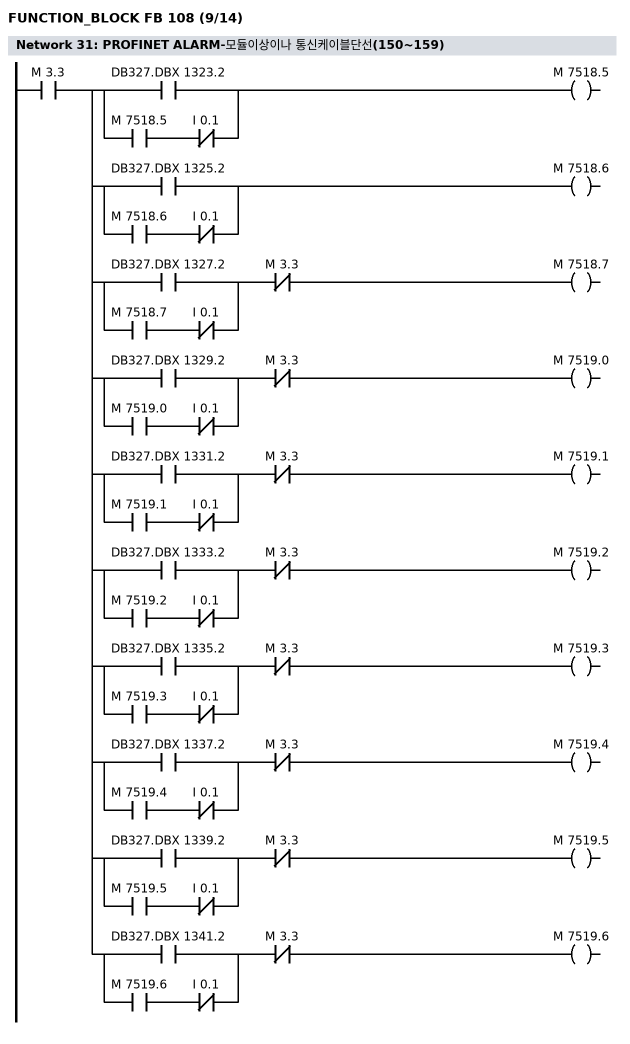

      A     M      3.3;
      =     L      0.0;
      A     L      0.0;
      A(    ;
      O     DB327.DBX 1323.2;
      O     ;
      A     M   7518.5;
      AN    I      0.1;
      )     ;
      =     M   7518.5;
      A     L      0.0;
      A(    ;
      O     DB327.DBX 1325.2;
      O     ;
      A     M   7518.6;
      AN    I      0.1;
      )     ;
      =     M   7518.6;
      A     L      0.0;
      A(    ;
      O     DB327.DBX 1327.2;
      O     ;
      A     M   7518.7;
      AN    I      0.1;
      )     ;
      AN    M      3.3;
      =     M   7518.7;
      A     L      0.0;
      A(    ;
      O     DB327.DBX 1329.2;
      O     ;
      A     M   7519.0;
      AN    I      0.1;
      )     ;
      AN    M      3.3;
      =     M   7519.0;
      A     L      0.0;
      A(    ;
      O     DB327.DBX 1331.2;
      O     ;
      A     M   7519.1;
      AN    I      0.1;
      )     ;
      AN    M      3.3;
      =     M   7519.1;
      A     L      0.0;
      A(    ;
      O     DB327.DBX 1333.2;
      O     ;
      A     M   7519.2;
      AN    I      0.1;
      )     ;
      AN    M      3.3;
      =     M   7519.2;
      A     L      0.0;
      A(    ;
      O     DB327.DBX 1335.2;
      O     ;
      A     M   7519.3;
      AN    I      0.1;
      )     ;
      AN    M      3.3;
      =     M   7519.3;
      A     L      0.0;
      A(    ;
      O     DB327.DBX 1337.2;
      O     ;
      A     M   7519.4;
      AN    I      0.1;
      )     ;
      AN    M      3.3;
      =     M   7519.4;
      A     L      0.0;
      A(    ;
      O     DB327.DBX 1339.2;
      O     ;
      A     M   7519.5;
      AN    I      0.1;
      )     ;
      AN    M      3.3;
      =     M   7519.5;
      A     L      0.0;
      A(    ;
      O     DB327.DBX 1341.2;
      O     ;
      A     M   7519.6;
      AN    I      0.1;
      )     ;
      AN    M      3.3;
      =     M   7519.6;
NETWORK
TITLE =PROFINET MODULE ERROR(1~10)
//
//
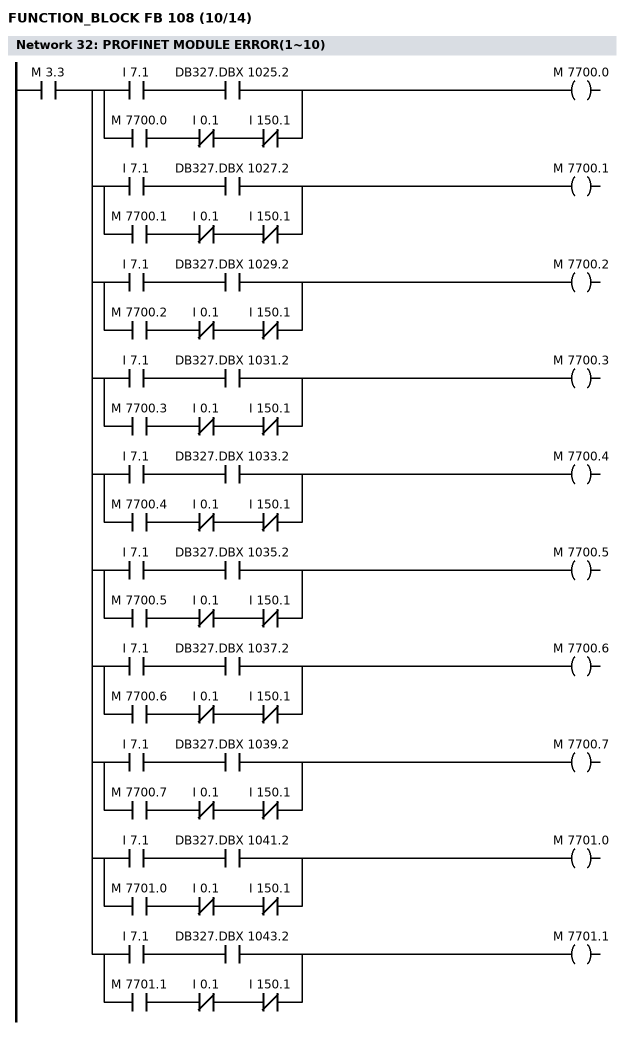
      A     M      3.3;
      =     L      0.0;
      A     L      0.0;
      A(    ;
      A     I      7.1;
      A     DB327.DBX 1025.2;
      O     ;
      A     M   7700.0;
      AN    I      0.1;
      AN    I    150.1;
      )     ;
      =     M   7700.0;
      A     L      0.0;
      A(    ;
      A     I      7.1;
      A     DB327.DBX 1027.2;
      O     ;
      A     M   7700.1;
      AN    I      0.1;
      AN    I    150.1;
      )     ;
      =     M   7700.1;
      A     L      0.0;
      A(    ;
      A     I      7.1;
      A     DB327.DBX 1029.2;
      O     ;
      A     M   7700.2;
      AN    I      0.1;
      AN    I    150.1;
      )     ;
      =     M   7700.2;
      A     L      0.0;
      A(    ;
      A     I      7.1;
      A     DB327.DBX 1031.2;
      O     ;
      A     M   7700.3;
      AN    I      0.1;
      AN    I    150.1;
      )     ;
      =     M   7700.3;
      A     L      0.0;
      A(    ;
      A     I      7.1;
      A     DB327.DBX 1033.2;
      O     ;
      A     M   7700.4;
      AN    I      0.1;
      AN    I    150.1;
      )     ;
      =     M   7700.4;
      A     L      0.0;
      A(    ;
      A     I      7.1;
      A     DB327.DBX 1035.2;
      O     ;
      A     M   7700.5;
      AN    I      0.1;
      AN    I    150.1;
      )     ;
      =     M   7700.5;
      A     L      0.0;
      A(    ;
      A     I      7.1;
      A     DB327.DBX 1037.2;
      O     ;
      A     M   7700.6;
      AN    I      0.1;
      AN    I    150.1;
      )     ;
      =     M   7700.6;
      A     L      0.0;
      A(    ;
      A     I      7.1;
      A     DB327.DBX 1039.2;
      O     ;
      A     M   7700.7;
      AN    I      0.1;
      AN    I    150.1;
      )     ;
      =     M   7700.7;
      A     L      0.0;
      A(    ;
      A     I      7.1;
      A     DB327.DBX 1041.2;
      O     ;
      A     M   7701.0;
      AN    I      0.1;
      AN    I    150.1;
      )     ;
      =     M   7701.0;
      A     L      0.0;
      A(    ;
      A     I      7.1;
      A     DB327.DBX 1043.2;
      O     ;
      A     M   7701.1;
      AN    I      0.1;
      AN    I    150.1;
      )     ;
      =     M   7701.1;
NETWORK
TITLE =PROFINET MODULE ERROR(11~20)
//
//
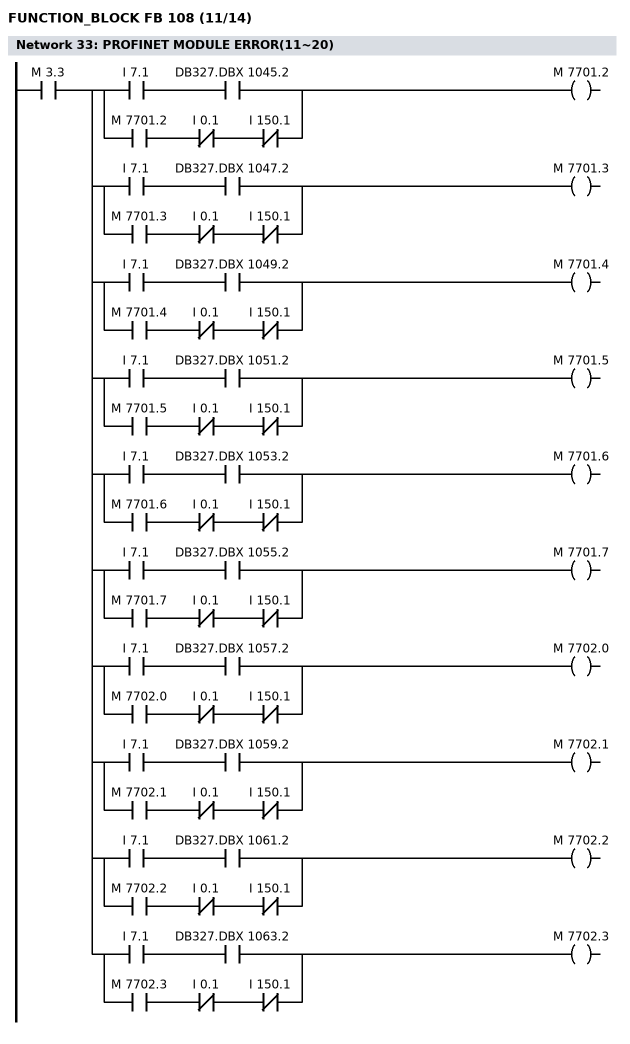
      A     M      3.3;
      =     L      0.0;
      A     L      0.0;
      A(    ;
      A     I      7.1;
      A     DB327.DBX 1045.2;
      O     ;
      A     M   7701.2;
      AN    I      0.1;
      AN    I    150.1;
      )     ;
      =     M   7701.2;
      A     L      0.0;
      A(    ;
      A     I      7.1;
      A     DB327.DBX 1047.2;
      O     ;
      A     M   7701.3;
      AN    I      0.1;
      AN    I    150.1;
      )     ;
      =     M   7701.3;
      A     L      0.0;
      A(    ;
      A     I      7.1;
      A     DB327.DBX 1049.2;
      O     ;
      A     M   7701.4;
      AN    I      0.1;
      AN    I    150.1;
      )     ;
      =     M   7701.4;
      A     L      0.0;
      A(    ;
      A     I      7.1;
      A     DB327.DBX 1051.2;
      O     ;
      A     M   7701.5;
      AN    I      0.1;
      AN    I    150.1;
      )     ;
      =     M   7701.5;
      A     L      0.0;
      A(    ;
      A     I      7.1;
      A     DB327.DBX 1053.2;
      O     ;
      A     M   7701.6;
      AN    I      0.1;
      AN    I    150.1;
      )     ;
      =     M   7701.6;
      A     L      0.0;
      A(    ;
      A     I      7.1;
      A     DB327.DBX 1055.2;
      O     ;
      A     M   7701.7;
      AN    I      0.1;
      AN    I    150.1;
      )     ;
      =     M   7701.7;
      A     L      0.0;
      A(    ;
      A     I      7.1;
      A     DB327.DBX 1057.2;
      O     ;
      A     M   7702.0;
      AN    I      0.1;
      AN    I    150.1;
      )     ;
      =     M   7702.0;
      A     L      0.0;
      A(    ;
      A     I      7.1;
      A     DB327.DBX 1059.2;
      O     ;
      A     M   7702.1;
      AN    I      0.1;
      AN    I    150.1;
      )     ;
      =     M   7702.1;
      A     L      0.0;
      A(    ;
      A     I      7.1;
      A     DB327.DBX 1061.2;
      O     ;
      A     M   7702.2;
      AN    I      0.1;
      AN    I    150.1;
      )     ;
      =     M   7702.2;
      A     L      0.0;
      A(    ;
      A     I      7.1;
      A     DB327.DBX 1063.2;
      O     ;
      A     M   7702.3;
      AN    I      0.1;
      AN    I    150.1;
      )     ;
      =     M   7702.3;
NETWORK
TITLE =PROFINET MODULE ERROR(21~30)
//
//
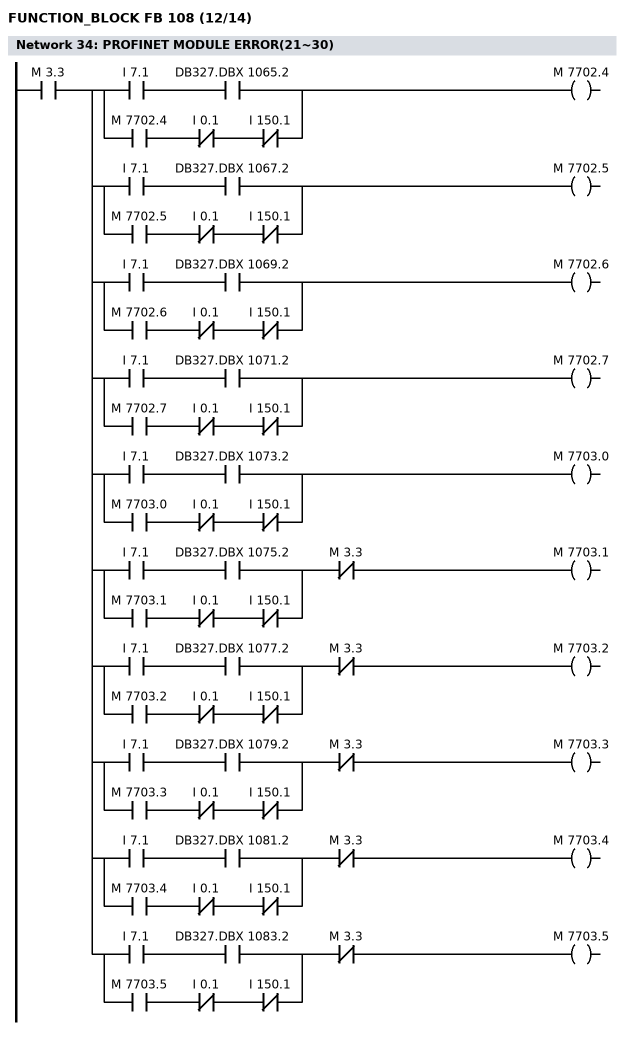
      A     M      3.3;
      =     L      0.0;
      A     L      0.0;
      A(    ;
      A     I      7.1;
      A     DB327.DBX 1065.2;
      O     ;
      A     M   7702.4;
      AN    I      0.1;
      AN    I    150.1;
      )     ;
      =     M   7702.4;
      A     L      0.0;
      A(    ;
      A     I      7.1;
      A     DB327.DBX 1067.2;
      O     ;
      A     M   7702.5;
      AN    I      0.1;
      AN    I    150.1;
      )     ;
      =     M   7702.5;
      A     L      0.0;
      A(    ;
      A     I      7.1;
      A     DB327.DBX 1069.2;
      O     ;
      A     M   7702.6;
      AN    I      0.1;
      AN    I    150.1;
      )     ;
      =     M   7702.6;
      A     L      0.0;
      A(    ;
      A     I      7.1;
      A     DB327.DBX 1071.2;
      O     ;
      A     M   7702.7;
      AN    I      0.1;
      AN    I    150.1;
      )     ;
      =     M   7702.7;
      A     L      0.0;
      A(    ;
      A     I      7.1;
      A     DB327.DBX 1073.2;
      O     ;
      A     M   7703.0;
      AN    I      0.1;
      AN    I    150.1;
      )     ;
      =     M   7703.0;
      A     L      0.0;
      A(    ;
      A     I      7.1;
      A     DB327.DBX 1075.2;
      O     ;
      A     M   7703.1;
      AN    I      0.1;
      AN    I    150.1;
      )     ;
      AN    M      3.3;
      =     M   7703.1;
      A     L      0.0;
      A(    ;
      A     I      7.1;
      A     DB327.DBX 1077.2;
      O     ;
      A     M   7703.2;
      AN    I      0.1;
      AN    I    150.1;
      )     ;
      AN    M      3.3;
      =     M   7703.2;
      A     L      0.0;
      A(    ;
      A     I      7.1;
      A     DB327.DBX 1079.2;
      O     ;
      A     M   7703.3;
      AN    I      0.1;
      AN    I    150.1;
      )     ;
      AN    M      3.3;
      =     M   7703.3;
      A     L      0.0;
      A(    ;
      A     I      7.1;
      A     DB327.DBX 1081.2;
      O     ;
      A     M   7703.4;
      AN    I      0.1;
      AN    I    150.1;
      )     ;
      AN    M      3.3;
      =     M   7703.4;
      A     L      0.0;
      A(    ;
      A     I      7.1;
      A     DB327.DBX 1083.2;
      O     ;
      A     M   7703.5;
      AN    I      0.1;
      AN    I    150.1;
      )     ;
      AN    M      3.3;
      =     M   7703.5;
NETWORK
TITLE =PROFINET MODULE ERROR(31~40)
//
//
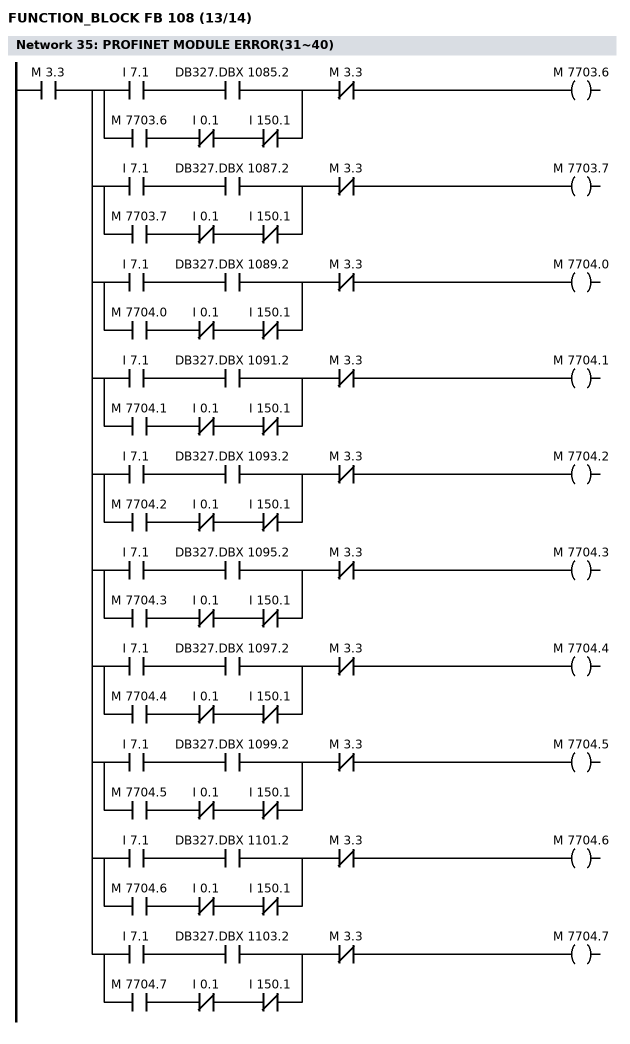
      A     M      3.3;
      =     L      0.0;
      A     L      0.0;
      A(    ;
      A     I      7.1;
      A     DB327.DBX 1085.2;
      O     ;
      A     M   7703.6;
      AN    I      0.1;
      AN    I    150.1;
      )     ;
      AN    M      3.3;
      =     M   7703.6;
      A     L      0.0;
      A(    ;
      A     I      7.1;
      A     DB327.DBX 1087.2;
      O     ;
      A     M   7703.7;
      AN    I      0.1;
      AN    I    150.1;
      )     ;
      AN    M      3.3;
      =     M   7703.7;
      A     L      0.0;
      A(    ;
      A     I      7.1;
      A     DB327.DBX 1089.2;
      O     ;
      A     M   7704.0;
      AN    I      0.1;
      AN    I    150.1;
      )     ;
      AN    M      3.3;
      =     M   7704.0;
      A     L      0.0;
      A(    ;
      A     I      7.1;
      A     DB327.DBX 1091.2;
      O     ;
      A     M   7704.1;
      AN    I      0.1;
      AN    I    150.1;
      )     ;
      AN    M      3.3;
      =     M   7704.1;
      A     L      0.0;
      A(    ;
      A     I      7.1;
      A     DB327.DBX 1093.2;
      O     ;
      A     M   7704.2;
      AN    I      0.1;
      AN    I    150.1;
      )     ;
      AN    M      3.3;
      =     M   7704.2;
      A     L      0.0;
      A(    ;
      A     I      7.1;
      A     DB327.DBX 1095.2;
      O     ;
      A     M   7704.3;
      AN    I      0.1;
      AN    I    150.1;
      )     ;
      AN    M      3.3;
      =     M   7704.3;
      A     L      0.0;
      A(    ;
      A     I      7.1;
      A     DB327.DBX 1097.2;
      O     ;
      A     M   7704.4;
      AN    I      0.1;
      AN    I    150.1;
      )     ;
      AN    M      3.3;
      =     M   7704.4;
      A     L      0.0;
      A(    ;
      A     I      7.1;
      A     DB327.DBX 1099.2;
      O     ;
      A     M   7704.5;
      AN    I      0.1;
      AN    I    150.1;
      )     ;
      AN    M      3.3;
      =     M   7704.5;
      A     L      0.0;
      A(    ;
      A     I      7.1;
      A     DB327.DBX 1101.2;
      O     ;
      A     M   7704.6;
      AN    I      0.1;
      AN    I    150.1;
      )     ;
      AN    M      3.3;
      =     M   7704.6;
      A     L      0.0;
      A(    ;
      A     I      7.1;
      A     DB327.DBX 1103.2;
      O     ;
      A     M   7704.7;
      AN    I      0.1;
      AN    I    150.1;
      )     ;
      AN    M      3.3;
      =     M   7704.7;
NETWORK
TITLE =PROFINET MODULE ERROR(150~159)
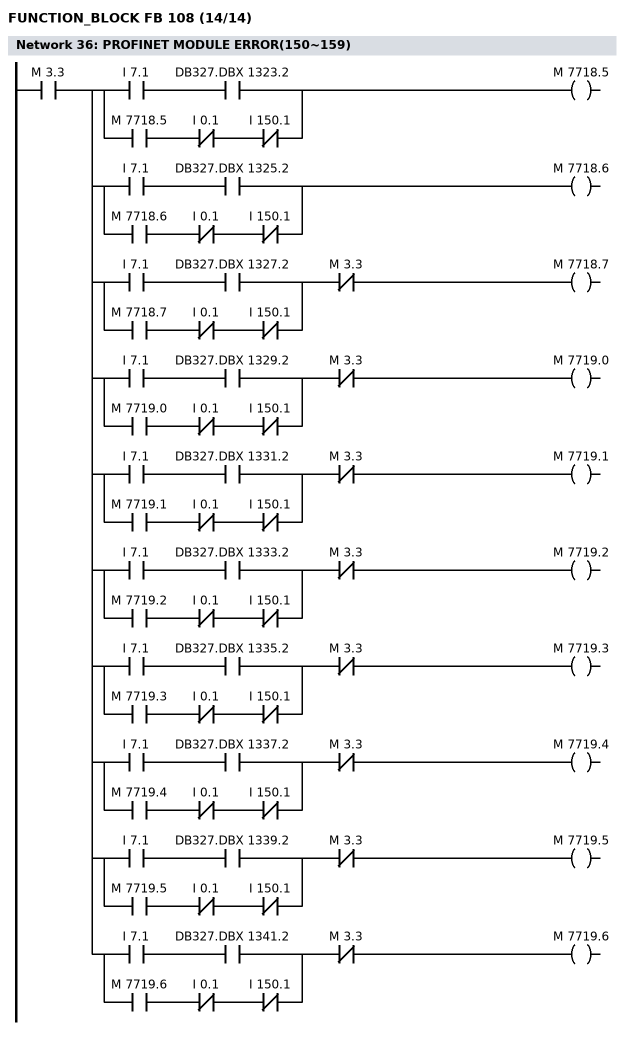

      A     M      3.3;
      =     L      0.0;
      A     L      0.0;
      A(    ;
      A     I      7.1;
      A     DB327.DBX 1323.2;
      O     ;
      A     M   7718.5;
      AN    I      0.1;
      AN    I    150.1;
      )     ;
      =     M   7718.5;
      A     L      0.0;
      A(    ;
      A     I      7.1;
      A     DB327.DBX 1325.2;
      O     ;
      A     M   7718.6;
      AN    I      0.1;
      AN    I    150.1;
      )     ;
      =     M   7718.6;
      A     L      0.0;
      A(    ;
      A     I      7.1;
      A     DB327.DBX 1327.2;
      O     ;
      A     M   7718.7;
      AN    I      0.1;
      AN    I    150.1;
      )     ;
      AN    M      3.3;
      =     M   7718.7;
      A     L      0.0;
      A(    ;
      A     I      7.1;
      A     DB327.DBX 1329.2;
      O     ;
      A     M   7719.0;
      AN    I      0.1;
      AN    I    150.1;
      )     ;
      AN    M      3.3;
      =     M   7719.0;
      A     L      0.0;
      A(    ;
      A     I      7.1;
      A     DB327.DBX 1331.2;
      O     ;
      A     M   7719.1;
      AN    I      0.1;
      AN    I    150.1;
      )     ;
      AN    M      3.3;
      =     M   7719.1;
      A     L      0.0;
      A(    ;
      A     I      7.1;
      A     DB327.DBX 1333.2;
      O     ;
      A     M   7719.2;
      AN    I      0.1;
      AN    I    150.1;
      )     ;
      AN    M      3.3;
      =     M   7719.2;
      A     L      0.0;
      A(    ;
      A     I      7.1;
      A     DB327.DBX 1335.2;
      O     ;
      A     M   7719.3;
      AN    I      0.1;
      AN    I    150.1;
      )     ;
      AN    M      3.3;
      =     M   7719.3;
      A     L      0.0;
      A(    ;
      A     I      7.1;
      A     DB327.DBX 1337.2;
      O     ;
      A     M   7719.4;
      AN    I      0.1;
      AN    I    150.1;
      )     ;
      AN    M      3.3;
      =     M   7719.4;
      A     L      0.0;
      A(    ;
      A     I      7.1;
      A     DB327.DBX 1339.2;
      O     ;
      A     M   7719.5;
      AN    I      0.1;
      AN    I    150.1;
      )     ;
      AN    M      3.3;
      =     M   7719.5;
      A     L      0.0;
      A(    ;
      A     I      7.1;
      A     DB327.DBX 1341.2;
      O     ;
      A     M   7719.6;
      AN    I      0.1;
      AN    I    150.1;
      )     ;
      AN    M      3.3;
      =     M   7719.6;
END_FUNCTION_BLOCK

DATA_BLOCK DB 108
TITLE =
VERSION : 0.0

 FB 108
BEGIN
END_DATA_BLOCK

FUNCTION FC 108 : VOID
TITLE =
VERSION : 0.1

BEGIN
NETWORK
TITLE =

      AN    OV;
      =     L      0.0;
      A     L      0.0;
      AN    M   1000.0;
      =     M   3800.0;
      A     L      0.0;
      AN    M   2500.0;
      =     M   3800.1;
      A     L      0.0;
      AN    I     16.0;
      =     M   3800.2;
      A     L      0.0;
      A     M    503.1;
      =     M   3800.3;
NETWORK
TITLE =

      AN    OV;
      =     L      0.0;
      A     L      0.0;
      A     M    503.3;
      =     M   3800.4;
      A     L      0.0;
      A     M    503.2;
      =     M   3800.5;
      A     L      0.0;
      A     M    503.2;
      =     M   3800.6;
      A     L      0.0;
      AN    I    100.7;
      =     M   3800.7;
NETWORK
TITLE =

      AN    OV;
      =     L      0.0;
      A     L      0.0;
      AN    I    100.3;
      =     M   3801.0;
      A     L      0.0;
      AN    I    100.1;
      =     M   3801.1;
      A     L      0.0;
      AN    I    100.6;
      =     M   3801.2;
      A     L      0.0;
      AN    I    100.4;
      =     M   3801.3;
NETWORK
TITLE =

      AN    OV;
      =     L      0.0;
      A     L      0.0;
      AN    I    100.0;
      =     M   3801.4;
      A     L      0.0;
      AN    I     29.5;
      =     M   3801.5;
      A     L      0.0;
      AN    I    129.1;
      =     M   3801.6;
      A     L      0.0;
      AN    I    100.2;
      =     M   3801.7;
NETWORK
TITLE =

      AN    OV;
      =     L      0.0;
      A     L      0.0;
      A     M   2503.4;
      =     M   3802.3;
      A     L      0.0;
      A     M   2503.5;
      =     M   3802.4;
      A     L      0.0;
      A     M   2503.6;
      =     M   3802.5;
      A     L      0.0;
      A     M   1003.6;
      =     M   3802.6;
      A     L      0.0;
      A     M   1004.2;
      =     M   3802.7;
NETWORK
TITLE =

      AN    OV;
      =     L      0.0;
      A     L      0.0;
      A     M   2504.2;
      =     M   3803.0;
      A     L      0.0;
      A(    ;
      O     M   2550.0;
      O     M   2550.1;
      )     ;
      =     M   3803.1;
      A     L      0.0;
      A(    ;
      O     M   2550.2;
      O     M   2550.3;
      )     ;
      =     M   3803.2;
      A     L      0.0;
      A(    ;
      O     M   2515.2;
      O     M   2550.4;
      O     M   2550.5;
      )     ;
      =     M   3803.3;
NETWORK
TITLE =

      AN    OV;
      =     L      0.0;
      A     L      0.0;
      A(    ;
      O     M   1050.0;
      O     M   1050.1;
      )     ;
      =     M   3803.4;
      A     L      0.0;
      A(    ;
      O     M   1050.2;
      O     M   1050.3;
      )     ;
      =     M   3803.5;
      A     L      0.0;
      A(    ;
      O     M   1050.4;
      O     M   1050.5;
      )     ;
      =     M   3803.6;
      A     L      0.0;
      A(    ;
      O     M   1050.6;
      O     M   1050.7;
      )     ;
      =     M   3803.7;
NETWORK
TITLE =

      AN    OV;
      =     L      0.0;
      A     L      0.0;
      A(    ;
      O     M   1051.0;
      O     M   1051.1;
      )     ;
      =     M   3804.0;
      A     L      0.0;
      A(    ;
      O     M   1051.2;
      O     M   1051.3;
      )     ;
      =     M   3804.1;
      A     L      0.0;
      A(    ;
      O     M   1051.4;
      O     M   1051.5;
      )     ;
      =     M   3804.2;
      A     L      0.0;
      A(    ;
      O     M   1051.6;
      O     M   1051.7;
      )     ;
      =     M   3804.3;
      A     L      0.0;
      A     M   5200.7;
      =     M   3805.5;
NETWORK
TITLE =
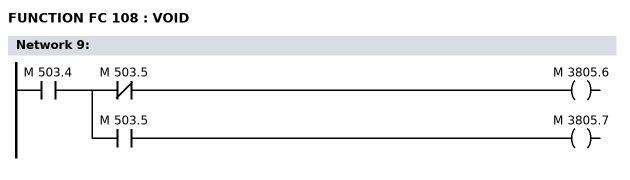

      A     M    503.4;
      =     L      0.0;
      A     L      0.0;
      AN    M    503.5;
      =     M   3805.6;
      A     L      0.0;
      A     M    503.5;
      =     M   3805.7;
NETWORK
TITLE =

      AN    OV;
      =     L      0.0;
      A     L      0.0;
      A(    ;
      O     I      2.1;
      O     I     49.6;
      O     T    134;
      )     ;
      =     M   3808.5;
      A     L      0.0;
      A     I      2.1;
      =     M   3808.6;
NETWORK
TITLE =
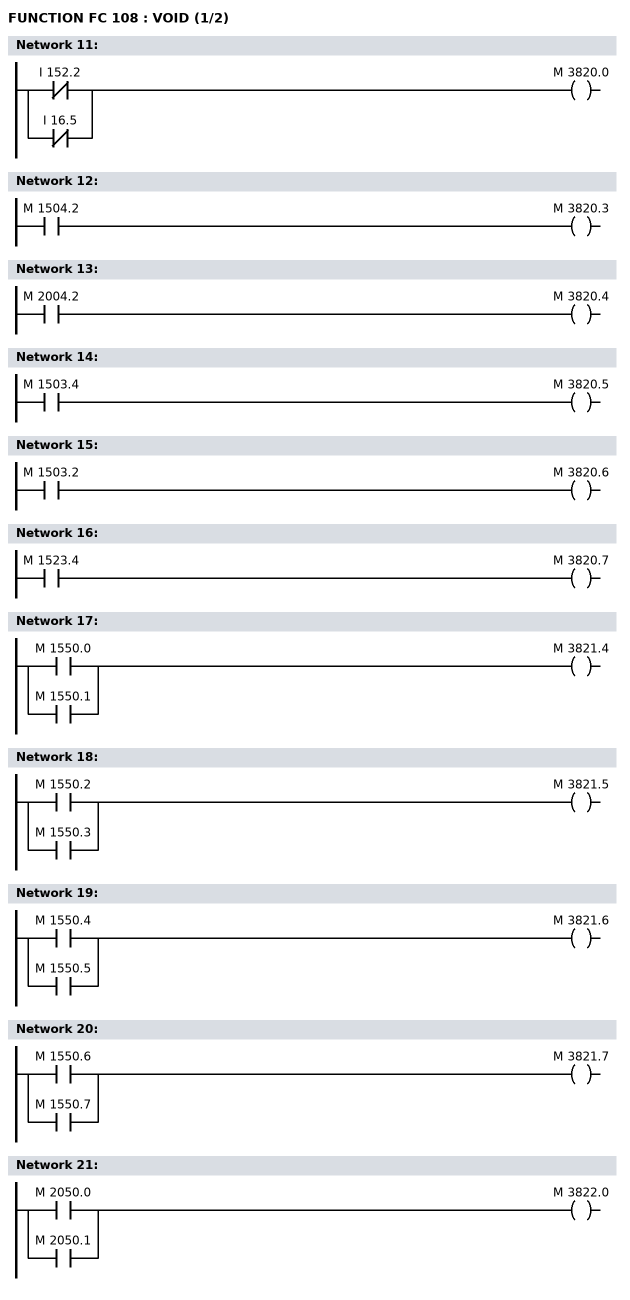

      ON    I    152.2;
      ON    I     16.5;
      =     M   3820.0;
NETWORK
TITLE =

      A     M   1504.2;
      =     M   3820.3;
NETWORK
TITLE =

      A     M   2004.2;
      =     M   3820.4;
NETWORK
TITLE =

      A     M   1503.4;
      =     M   3820.5;
NETWORK
TITLE =

      A     M   1503.2;
      =     M   3820.6;
NETWORK
TITLE =

      A     M   1523.4;
      =     M   3820.7;
NETWORK
TITLE =

      O     M   1550.0;
      O     M   1550.1;
      =     M   3821.4;
NETWORK
TITLE =

      O     M   1550.2;
      O     M   1550.3;
      =     M   3821.5;
NETWORK
TITLE =

      O     M   1550.4;
      O     M   1550.5;
      =     M   3821.6;
NETWORK
TITLE =

      O     M   1550.6;
      O     M   1550.7;
      =     M   3821.7;
NETWORK
TITLE =

      O     M   2050.0;
      O     M   2050.1;
      =     M   3822.0;
NETWORK
TITLE =
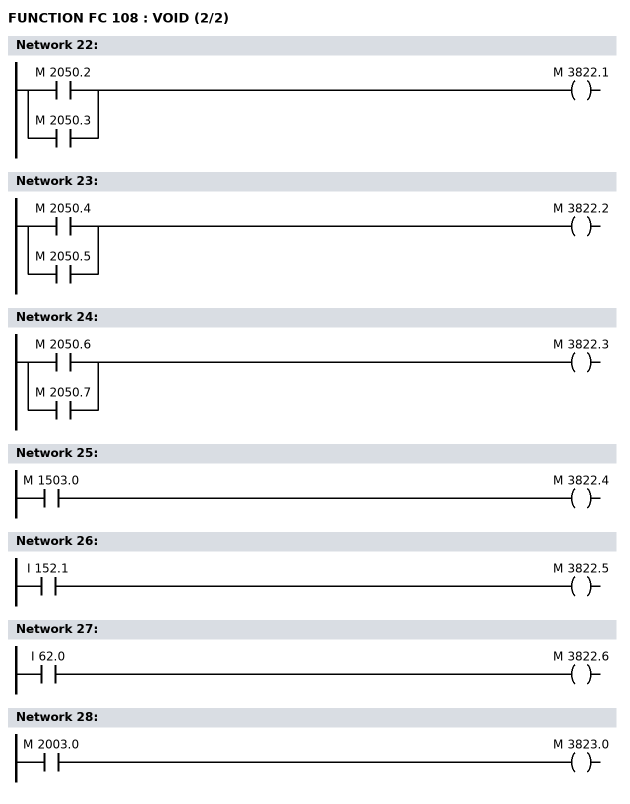

      O     M   2050.2;
      O     M   2050.3;
      =     M   3822.1;
NETWORK
TITLE =

      O     M   2050.4;
      O     M   2050.5;
      =     M   3822.2;
NETWORK
TITLE =

      O     M   2050.6;
      O     M   2050.7;
      =     M   3822.3;
NETWORK
TITLE =

      A     M   1503.0;
      =     M   3822.4;
NETWORK
TITLE =

      A     I    152.1;
      =     M   3822.5;
NETWORK
TITLE =

      A     I     62.0;
      =     M   3822.6;
NETWORK
TITLE =

      A     M   2003.0;
      =     M   3823.0;
NETWORK
TITLE =

      AN    OV;
      =     L      0.0;
      A     L      0.0;
      AN    I   1011.0;
      =     M   3824.0;
      A     L      0.0;
      A     I   1011.1;
      =     M   3824.1;
      A     L      0.0;
      A     I   1011.2;
      =     M   3824.2;
      A     L      0.0;
      A     I   1011.4;
      =     M   3824.3;
      A     L      0.0;
      A     I   1011.5;
      =     M   3824.4;
      A     L      0.0;
      A     I   1011.6;
      =     M   3824.5;
      A     L      0.0;
      A     I   1011.7;
      =     M   3824.6;
      A     L      0.0;
      A     I   1010.5;
      =     M   3824.7;
NETWORK
TITLE =

      AN    OV;
      =     L      0.0;
      A     L      0.0;
      AN    I   1019.0;
      =     M   3825.0;
      A     L      0.0;
      A     I   1019.1;
      =     M   3825.1;
      A     L      0.0;
      A     I   1019.2;
      =     M   3825.2;
      A     L      0.0;
      A     I   1019.4;
      =     M   3825.3;
      A     L      0.0;
      A     I   1019.5;
      =     M   3825.4;
      A     L      0.0;
      A     I   1019.6;
      =     M   3825.5;
      A     L      0.0;
      A     I   1019.7;
      =     M   3825.6;
      A     L      0.0;
      A     I   1018.5;
      =     M   3825.7;
NETWORK
TITLE =

      AN    OV;
      =     L      0.0;
      A     L      0.0;
      AN    I   1027.0;
      =     M   3826.0;
      A     L      0.0;
      A     I   1027.1;
      =     M   3826.1;
      A     L      0.0;
      A     I   1027.2;
      =     M   3826.2;
      A     L      0.0;
      A     I   1027.4;
      =     M   3826.3;
      A     L      0.0;
      A     I   1027.5;
      =     M   3826.4;
      A     L      0.0;
      A     I   1027.6;
      =     M   3826.5;
      A     L      0.0;
      A     I   1027.7;
      =     M   3826.6;
      A     L      0.0;
      A     I   1026.5;
      =     M   3826.7;
NETWORK
TITLE =

      AN    OV;
      =     L      0.0;
      A     L      0.0;
      AN    I   1035.0;
      =     M   3827.0;
      A     L      0.0;
      A     I   1035.1;
      =     M   3827.1;
      A     L      0.0;
      A     I   1035.2;
      =     M   3827.2;
      A     L      0.0;
      A     I   1035.4;
      =     M   3827.3;
      A     L      0.0;
      A     I   1035.5;
      =     M   3827.4;
      A     L      0.0;
      A     I   1035.6;
      =     M   3827.5;
      A     L      0.0;
      A     I   1035.7;
      =     M   3827.6;
      A     L      0.0;
      A     I   1034.5;
      =     M   3827.7;
NETWORK
TITLE =
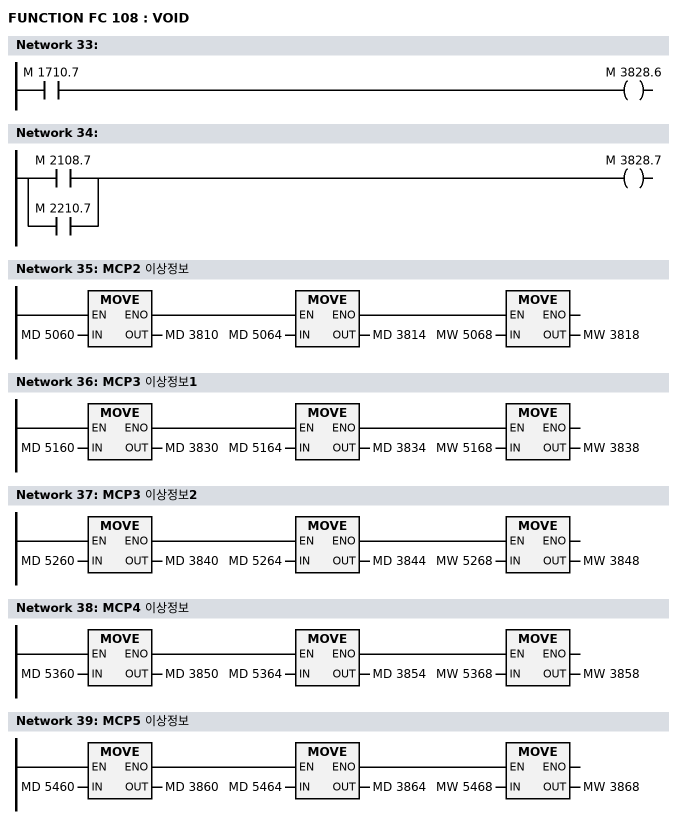

      A     M   1710.7;
      =     M   3828.6;
NETWORK
TITLE =

      O     M   2108.7;
      O     M   2210.7;
      =     M   3828.7;
NETWORK
TITLE =MCP2 이상정보

      A(    ;
      A(    ;
      L     MD  5060;
      T     MD  3810;
      SET   ;
      SAVE  ;
      CLR   ;
      A     BR;
      )     ;
      JNB   _001;
      L     MD  5064;
      T     MD  3814;
      SET   ;
      SAVE  ;
      CLR   ;
_001: A     BR;
      )     ;
      JNB   _002;
      L     MW  5068;
      T     MW  3818;
_002: NOP   0;
NETWORK
TITLE =MCP3 이상정보1

      A(    ;
      A(    ;
      L     MD  5160;
      T     MD  3830;
      SET   ;
      SAVE  ;
      CLR   ;
      A     BR;
      )     ;
      JNB   _003;
      L     MD  5164;
      T     MD  3834;
      SET   ;
      SAVE  ;
      CLR   ;
_003: A     BR;
      )     ;
      JNB   _004;
      L     MW  5168;
      T     MW  3838;
_004: NOP   0;
NETWORK
TITLE =MCP3 이상정보2

      A(    ;
      A(    ;
      L     MD  5260;
      T     MD  3840;
      SET   ;
      SAVE  ;
      CLR   ;
      A     BR;
      )     ;
      JNB   _005;
      L     MD  5264;
      T     MD  3844;
      SET   ;
      SAVE  ;
      CLR   ;
_005: A     BR;
      )     ;
      JNB   _006;
      L     MW  5268;
      T     MW  3848;
_006: NOP   0;
NETWORK
TITLE =MCP4 이상정보

      A(    ;
      A(    ;
      L     MD  5360;
      T     MD  3850;
      SET   ;
      SAVE  ;
      CLR   ;
      A     BR;
      )     ;
      JNB   _007;
      L     MD  5364;
      T     MD  3854;
      SET   ;
      SAVE  ;
      CLR   ;
_007: A     BR;
      )     ;
      JNB   _008;
      L     MW  5368;
      T     MW  3858;
_008: NOP   0;
NETWORK
TITLE =MCP5 이상정보

      A(    ;
      A(    ;
      L     MD  5460;
      T     MD  3860;
      SET   ;
      SAVE  ;
      CLR   ;
      A     BR;
      )     ;
      JNB   _009;
      L     MD  5464;
      T     MD  3864;
      SET   ;
      SAVE  ;
      CLR   ;
_009: A     BR;
      )     ;
      JNB   _00a;
      L     MW  5468;
      T     MW  3868;
_00a: NOP   0;
END_FUNCTION

FUNCTION FC 109 : VOID
TITLE =
VERSION : 0.1

BEGIN
NETWORK
TITLE =
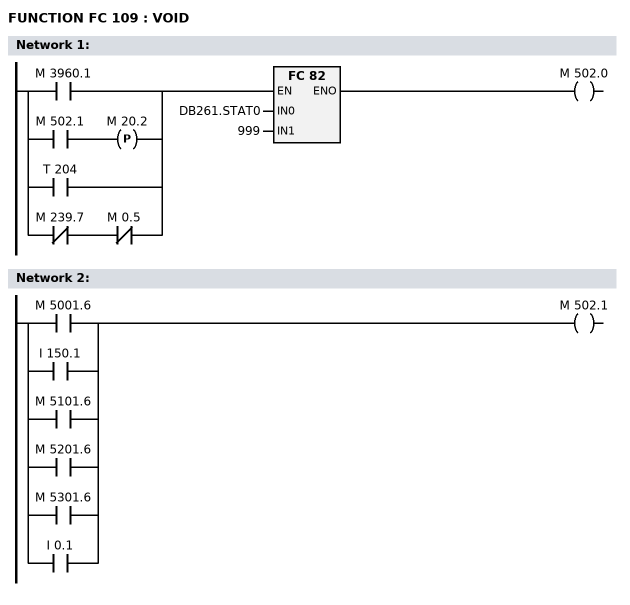

      A(    ;
      O     M   3960.1;
      O(    ;
      A     M    502.1;
      FP    M     20.2;
      )     ;
      O     T    204;
      O     ;
      AN    M    239.7;
      AN    M      0.5;
      )     ;
      JNB   _001;
      CALL FC    82 (
           IN0                      := DB261.STAT0,
           IN1                      := 999);
_001: A     BR;
      =     M    502.0;
NETWORK
TITLE =

      O     M   5001.6;
      O     I    150.1;
      O     M   5101.6;
      O     M   5201.6;
      O     M   5301.6;
      O     I      0.1;
      =     M    502.1;
NETWORK
TITLE =

      AN    OV;
      =     L      0.0;
      A     L      0.0;
      A     M    502.0;
      L     S5T#1S;
      SE    T    205;
      A     L      0.0;
      AN    M    239.7;
      L     S5T#1S;
      SD    T    203;
      A     L      0.0;
      A     T    203;
      L     S5T#1S;
      SE    T    204;
NETWORK
TITLE =
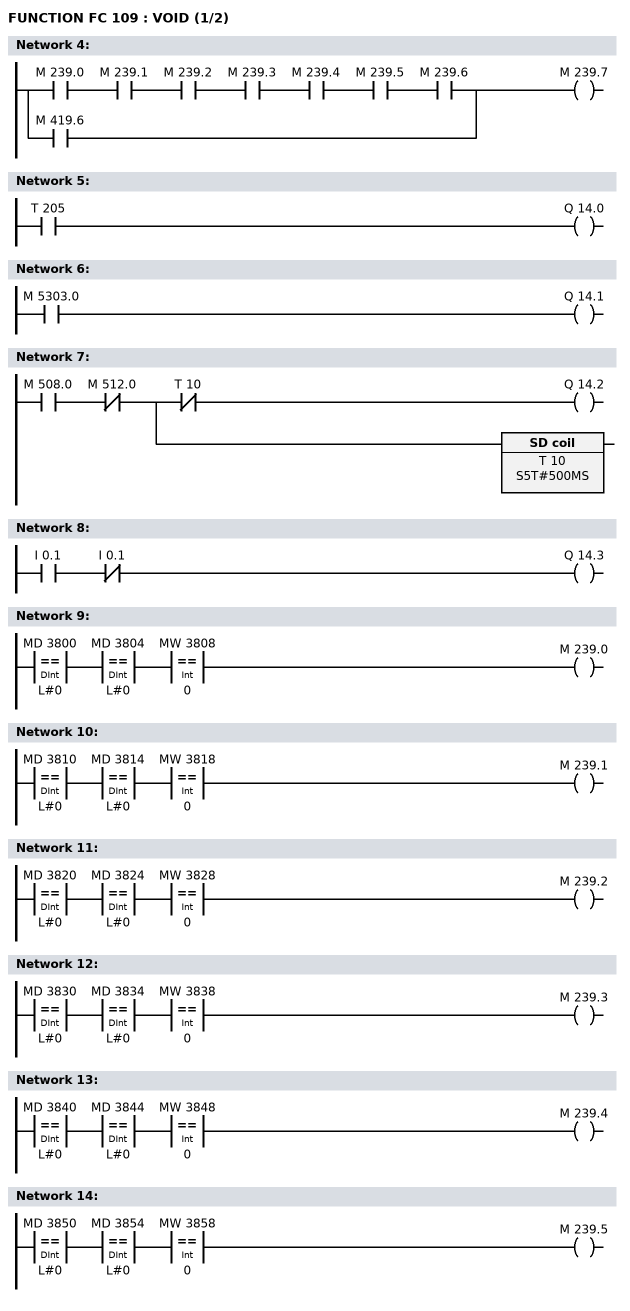

      A     M    239.0;
      A     M    239.1;
      A     M    239.2;
      A     M    239.3;
      A     M    239.4;
      A     M    239.5;
      A     M    239.6;
      O     M    419.6;
      =     M    239.7;
NETWORK
TITLE =

      A     T    205;
      =     Q     14.0;
NETWORK
TITLE =

      A     M   5303.0;
      =     Q     14.1;
NETWORK
TITLE =

      A     M    508.0;
      AN    M    512.0;
      =     L      0.0;
      A     L      0.0;
      AN    T     10;
      =     Q     14.2;
      A     L      0.0;
      BLD   102;
      L     S5T#500MS;
      SD    T     10;
NETWORK
TITLE =

      A     I      0.1;
      AN    I      0.1;
      =     Q     14.3;
NETWORK
TITLE =

      A(    ;
      L     MD  3800;
      L     L#0;
      ==D   ;
      )     ;
      A(    ;
      L     MD  3804;
      L     L#0;
      ==D   ;
      )     ;
      A(    ;
      L     MW  3808;
      L     0;
      ==I   ;
      )     ;
      =     M    239.0;
NETWORK
TITLE =

      A(    ;
      L     MD  3810;
      L     L#0;
      ==D   ;
      )     ;
      A(    ;
      L     MD  3814;
      L     L#0;
      ==D   ;
      )     ;
      A(    ;
      L     MW  3818;
      L     0;
      ==I   ;
      )     ;
      =     M    239.1;
NETWORK
TITLE =

      A(    ;
      L     MD  3820;
      L     L#0;
      ==D   ;
      )     ;
      A(    ;
      L     MD  3824;
      L     L#0;
      ==D   ;
      )     ;
      A(    ;
      L     MW  3828;
      L     0;
      ==I   ;
      )     ;
      =     M    239.2;
NETWORK
TITLE =

      A(    ;
      L     MD  3830;
      L     L#0;
      ==D   ;
      )     ;
      A(    ;
      L     MD  3834;
      L     L#0;
      ==D   ;
      )     ;
      A(    ;
      L     MW  3838;
      L     0;
      ==I   ;
      )     ;
      =     M    239.3;
NETWORK
TITLE =

      A(    ;
      L     MD  3840;
      L     L#0;
      ==D   ;
      )     ;
      A(    ;
      L     MD  3844;
      L     L#0;
      ==D   ;
      )     ;
      A(    ;
      L     MW  3848;
      L     0;
      ==I   ;
      )     ;
      =     M    239.4;
NETWORK
TITLE =

      A(    ;
      L     MD  3850;
      L     L#0;
      ==D   ;
      )     ;
      A(    ;
      L     MD  3854;
      L     L#0;
      ==D   ;
      )     ;
      A(    ;
      L     MW  3858;
      L     0;
      ==I   ;
      )     ;
      =     M    239.5;
NETWORK
TITLE =
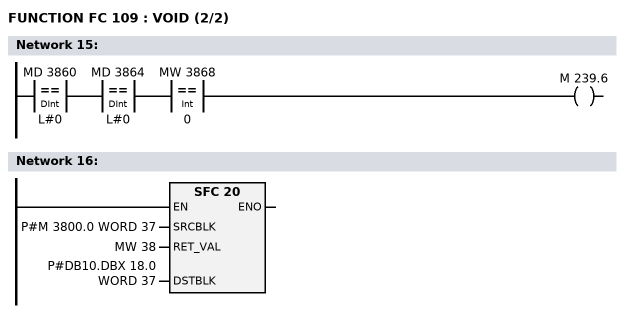

      A(    ;
      L     MD  3860;
      L     L#0;
      ==D   ;
      )     ;
      A(    ;
      L     MD  3864;
      L     L#0;
      ==D   ;
      )     ;
      A(    ;
      L     MW  3868;
      L     0;
      ==I   ;
      )     ;
      =     M    239.6;
NETWORK
TITLE =

      CALL SFC   20 (
           SRCBLK                   := P#M 3800.0 WORD 37,
           RET_VAL                  := MW    38,
           DSTBLK                   := P#DB10.DBX 18.0 WORD 37);
      NOP   0;
END_FUNCTION

FUNCTION_BLOCK FB 110
TITLE =
VERSION : 0.1


VAR
  S_SHUTTLE_MODE : FB 402;
END_VAR
BEGIN
NETWORK
TITLE =
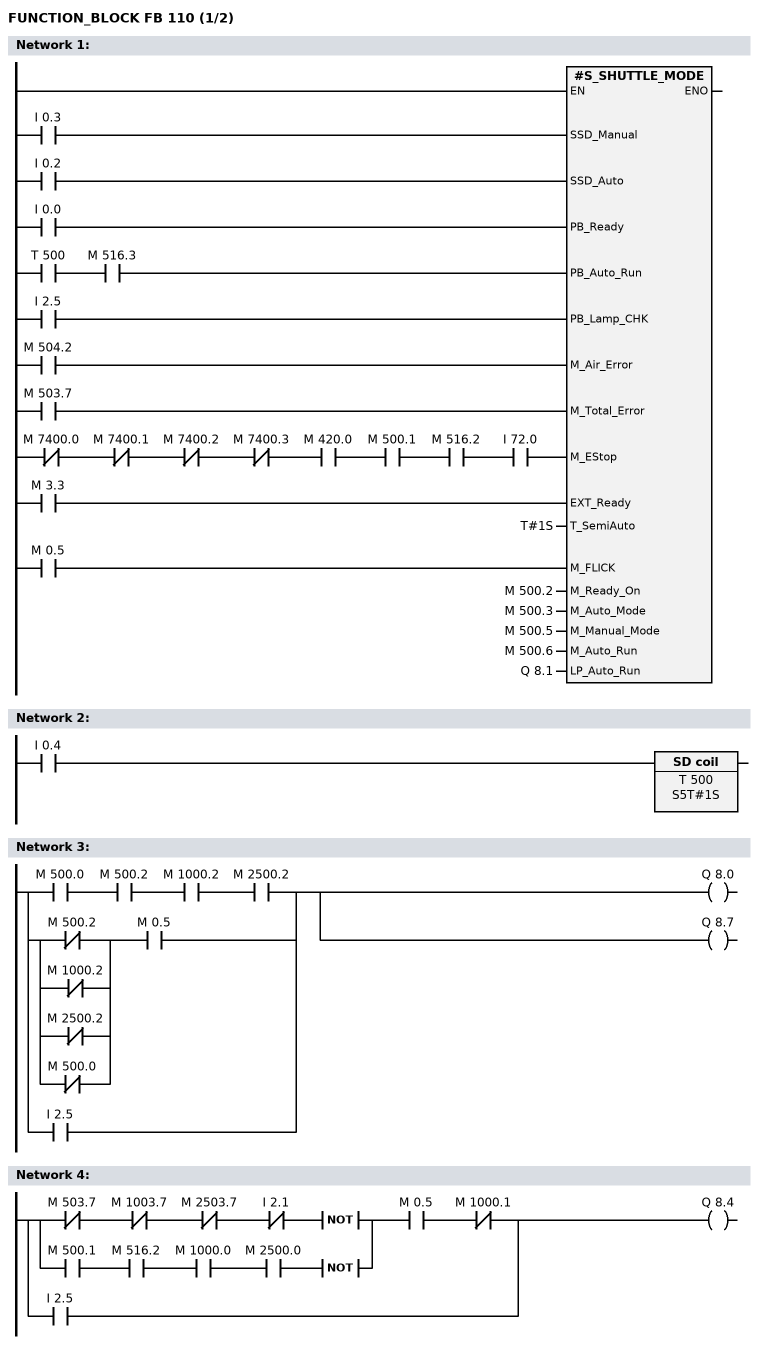

      A     I      0.3;
      =     L      0.0;
      BLD   103;
      A     I      0.2;
      =     L      0.1;
      BLD   103;
      A     I      0.0;
      =     L      0.2;
      BLD   103;
      A     T    500;
      A     M    516.3;
      =     L      0.3;
      BLD   103;
      A     I      2.5;
      =     L      0.6;
      BLD   103;
      A     M    504.2;
      =     L      0.7;
      BLD   103;
      A     M    503.7;
      =     L      1.1;
      BLD   103;
      AN    M   7400.0;
      AN    M   7400.1;
      AN    M   7400.2;
      AN    M   7400.3;
      A     M    420.0;
      A     M    500.1;
      A     M    516.2;
      A     I     72.0;
      =     L      1.2;
      BLD   103;
      A     M      3.3;
      =     L      1.3;
      BLD   103;
      A     M      0.5;
      =     L      1.5;
      BLD   103;
      CALL #S_SHUTTLE_MODE (
           SSD_Manual               := L      0.0,
           SSD_Auto                 := L      0.1,
           PB_Ready                 := L      0.2,
           PB_Auto_Run              := L      0.3,
           PB_Lamp_CHK              := L      0.6,
           M_Air_Error              := L      0.7,
           M_Total_Error            := L      1.1,
           M_EStop                  := L      1.2,
           EXT_Ready                := L      1.3,
           T_SemiAuto               := T#1S,
           M_FLICK                  := L      1.5,
           M_Ready_On               := M    500.2,
           M_Auto_Mode              := M    500.3,
           M_Manual_Mode            := M    500.5,
           M_Auto_Run               := M    500.6,
           LP_Auto_Run              := Q      8.1);
      NOP   0;
NETWORK
TITLE =

      A     I      0.4;
      L     S5T#1S;
      SD    T    500;
NETWORK
TITLE =

      A     M    500.0;
      A     M    500.2;
      A     M   1000.2;
      A     M   2500.2;
      O     ;
      A(    ;
      ON    M    500.2;
      ON    M   1000.2;
      ON    M   2500.2;
      ON    M    500.0;
      )     ;
      A     M      0.5;
      O     I      2.5;
      =     Q      8.0;
      =     Q      8.7;
NETWORK
TITLE =

      A(    ;
      AN    M    503.7;
      AN    M   1003.7;
      AN    M   2503.7;
      AN    I      2.1;
      NOT   ;
      O(    ;
      A     M    500.1;
      A     M    516.2;
      A     M   1000.0;
      A     M   2500.0;
      NOT   ;
      )     ;
      )     ;
      A     M      0.5;
      AN    M   1000.1;
      O     I      2.5;
      =     Q      8.4;
NETWORK
TITLE =
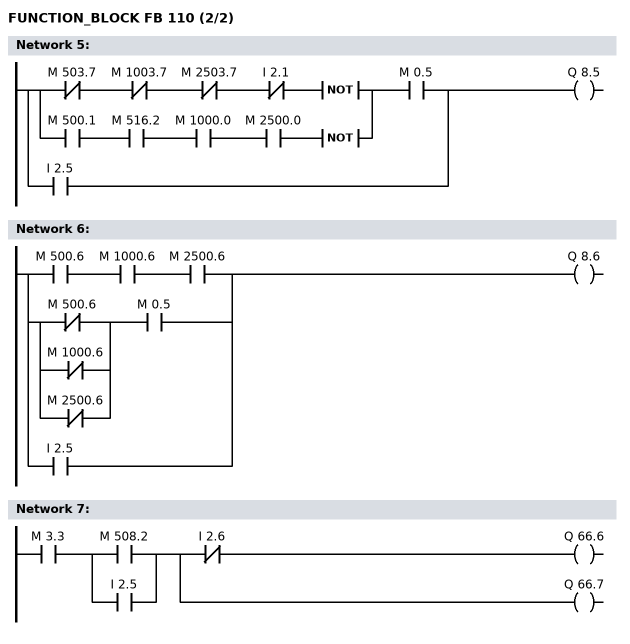

      A(    ;
      AN    M    503.7;
      AN    M   1003.7;
      AN    M   2503.7;
      AN    I      2.1;
      NOT   ;
      O(    ;
      A     M    500.1;
      A     M    516.2;
      A     M   1000.0;
      A     M   2500.0;
      NOT   ;
      )     ;
      )     ;
      A     M      0.5;
      O     I      2.5;
      =     Q      8.5;
NETWORK
TITLE =

      A     M    500.6;
      A     M   1000.6;
      A     M   2500.6;
      O     ;
      A(    ;
      ON    M    500.6;
      ON    M   1000.6;
      ON    M   2500.6;
      )     ;
      A     M      0.5;
      O     I      2.5;
      =     Q      8.6;
NETWORK
TITLE =

      A     M      3.3;
      A(    ;
      O     M    508.2;
      O     I      2.5;
      )     ;
      =     L      0.0;
      A     L      0.0;
      AN    I      2.6;
      =     Q     66.6;
      A     L      0.0;
      BLD   102;
      =     Q     66.7;
END_FUNCTION_BLOCK

DATA_BLOCK DB 110
TITLE =
VERSION : 0.0

 FB 110
BEGIN
   S_SHUTTLE_MODE.SSD_Manual := FALSE;
   S_SHUTTLE_MODE.SSD_Auto := FALSE;
   S_SHUTTLE_MODE.PB_Ready := FALSE;
   S_SHUTTLE_MODE.PB_Auto_Run := FALSE;
   S_SHUTTLE_MODE.PB_Remote_Ready := FALSE;
   S_SHUTTLE_MODE.PB_Remote_Auto_Run := FALSE;
   S_SHUTTLE_MODE.PB_Lamp_CHK := FALSE;
   S_SHUTTLE_MODE.M_Air_Error := FALSE;
   S_SHUTTLE_MODE.M_Water_Error := FALSE;
   S_SHUTTLE_MODE.M_Total_Error := FALSE;
   S_SHUTTLE_MODE.M_EStop := FALSE;
   S_SHUTTLE_MODE.EXT_Ready := FALSE;
   S_SHUTTLE_MODE.EXT_Auto := FALSE;
   S_SHUTTLE_MODE.T_SemiAuto := T#0MS;
   S_SHUTTLE_MODE.M_FLICK := FALSE;
   S_SHUTTLE_MODE.M_Ready_On := FALSE;
   S_SHUTTLE_MODE.M_Auto_Mode := FALSE;
   S_SHUTTLE_MODE.M_SemiAuto_Mode := FALSE;
   S_SHUTTLE_MODE.M_Manual_Mode := FALSE;
   S_SHUTTLE_MODE.M_Auto_Run := FALSE;
   S_SHUTTLE_MODE.LP_Ready_On := FALSE;
   S_SHUTTLE_MODE.LP_Auto_Run := FALSE;
   S_SHUTTLE_MODE.AUTO_MODE_DELAY.IN := FALSE;
   S_SHUTTLE_MODE.AUTO_MODE_DELAY.PT := T#0MS;
   S_SHUTTLE_MODE.AUTO_MODE_DELAY.Q := FALSE;
   S_SHUTTLE_MODE.AUTO_MODE_DELAY.ET := T#0MS;
   S_SHUTTLE_MODE.AUTO_MODE_DELAY.STATE := B#16#0;
   S_SHUTTLE_MODE.AUTO_MODE_DELAY.STIME := T#0MS;
   S_SHUTTLE_MODE.AUTO_MODE_DELAY.ATIME := T#0MS;
   S_SHUTTLE_MODE.SEMI_AUTO_DELAY.IN := FALSE;
   S_SHUTTLE_MODE.SEMI_AUTO_DELAY.PT := T#0MS;
   S_SHUTTLE_MODE.SEMI_AUTO_DELAY.Q := FALSE;
   S_SHUTTLE_MODE.SEMI_AUTO_DELAY.ET := T#0MS;
   S_SHUTTLE_MODE.SEMI_AUTO_DELAY.STATE := B#16#0;
   S_SHUTTLE_MODE.SEMI_AUTO_DELAY.STIME := T#0MS;
   S_SHUTTLE_MODE.SEMI_AUTO_DELAY.ATIME := T#0MS;
   S_SHUTTLE_MODE.MANUAL_DELAY.IN := FALSE;
   S_SHUTTLE_MODE.MANUAL_DELAY.PT := T#0MS;
   S_SHUTTLE_MODE.MANUAL_DELAY.Q := FALSE;
   S_SHUTTLE_MODE.MANUAL_DELAY.ET := T#0MS;
   S_SHUTTLE_MODE.MANUAL_DELAY.STATE := B#16#0;
   S_SHUTTLE_MODE.MANUAL_DELAY.STIME := T#0MS;
   S_SHUTTLE_MODE.MANUAL_DELAY.ATIME := T#0MS;
END_DATA_BLOCK

FUNCTION FC 110 : VOID
TITLE =
VERSION : 0.1

BEGIN
NETWORK
TITLE =
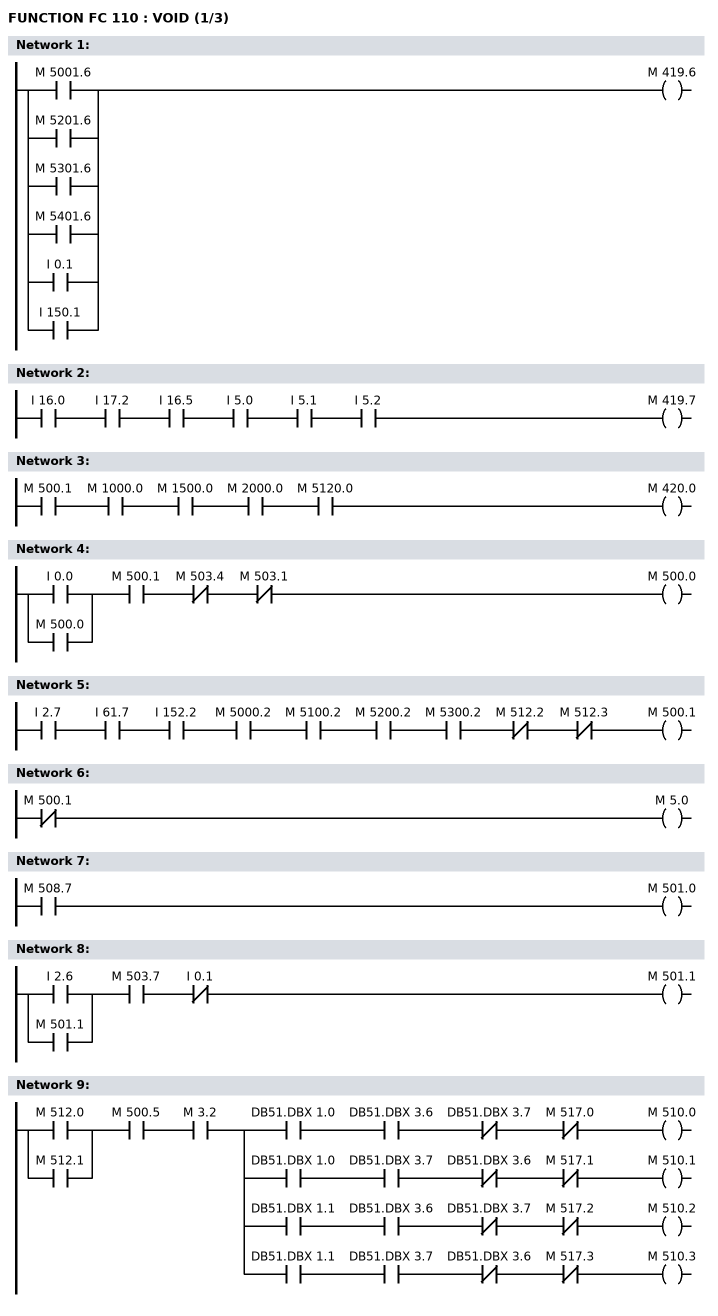

      O     M   5001.6;
      O     M   5201.6;
      O     M   5301.6;
      O     M   5401.6;
      O     I      0.1;
      O     I    150.1;
      =     M    419.6;
NETWORK
TITLE =

      A     I     16.0;
      A     I     17.2;
      A     I     16.5;
      A     I      5.0;
      A     I      5.1;
      A     I      5.2;
      =     M    419.7;
NETWORK
TITLE =

      A     M    500.1;
      A     M   1000.0;
      A     M   1500.0;
      A     M   2000.0;
      A     M   5120.0;
      =     M    420.0;
NETWORK
TITLE =

      A(    ;
      O     I      0.0;
      O     M    500.0;
      )     ;
      A     M    500.1;
      AN    M    503.4;
      AN    M    503.1;
      =     M    500.0;
NETWORK
TITLE =

      A     I      2.7;
      A     I     61.7;
      A     I    152.2;
      A     M   5000.2;
      A     M   5100.2;
      A     M   5200.2;
      A     M   5300.2;
      AN    M    512.2;
      AN    M    512.3;
      =     M    500.1;
NETWORK
TITLE =

      AN    M    500.1;
      =     M      5.0;
NETWORK
TITLE =

      A     M    508.7;
      =     M    501.0;
NETWORK
TITLE =

      A(    ;
      O     I      2.6;
      O     M    501.1;
      )     ;
      A     M    503.7;
      AN    I      0.1;
      =     M    501.1;
NETWORK
TITLE =

      A(    ;
      O     M    512.0;
      O     M    512.1;
      )     ;
      A     M    500.5;
      A     M      3.2;
      =     L      0.0;
      A     L      0.0;
      A     DB51.DBX    1.0;
      A     DB51.DBX    3.6;
      AN    DB51.DBX    3.7;
      AN    M    517.0;
      =     M    510.0;
      A     L      0.0;
      A     DB51.DBX    1.0;
      A     DB51.DBX    3.7;
      AN    DB51.DBX    3.6;
      AN    M    517.1;
      =     M    510.1;
      A     L      0.0;
      A     DB51.DBX    1.1;
      A     DB51.DBX    3.6;
      AN    DB51.DBX    3.7;
      AN    M    517.2;
      =     M    510.2;
      A     L      0.0;
      A     DB51.DBX    1.1;
      A     DB51.DBX    3.7;
      AN    DB51.DBX    3.6;
      AN    M    517.3;
      =     M    510.3;
NETWORK
TITLE =
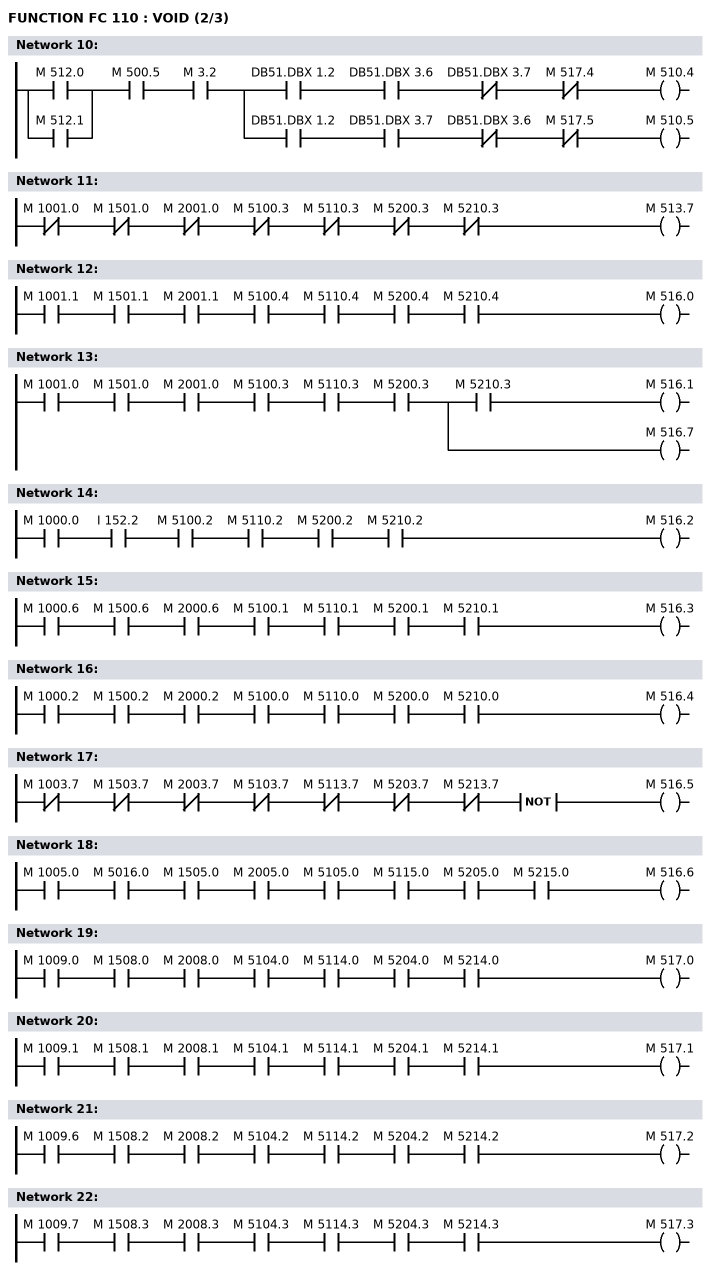

      A(    ;
      O     M    512.0;
      O     M    512.1;
      )     ;
      A     M    500.5;
      A     M      3.2;
      =     L      0.0;
      A     L      0.0;
      A     DB51.DBX    1.2;
      A     DB51.DBX    3.6;
      AN    DB51.DBX    3.7;
      AN    M    517.4;
      =     M    510.4;
      A     L      0.0;
      A     DB51.DBX    1.2;
      A     DB51.DBX    3.7;
      AN    DB51.DBX    3.6;
      AN    M    517.5;
      =     M    510.5;
NETWORK
TITLE =

      AN    M   1001.0;
      AN    M   1501.0;
      AN    M   2001.0;
      AN    M   5100.3;
      AN    M   5110.3;
      AN    M   5200.3;
      AN    M   5210.3;
      =     M    513.7;
NETWORK
TITLE =

      A     M   1001.1;
      A     M   1501.1;
      A     M   2001.1;
      A     M   5100.4;
      A     M   5110.4;
      A     M   5200.4;
      A     M   5210.4;
      =     M    516.0;
NETWORK
TITLE =

      A     M   1001.0;
      A     M   1501.0;
      A     M   2001.0;
      A     M   5100.3;
      A     M   5110.3;
      A     M   5200.3;
      =     L      0.0;
      A     L      0.0;
      A     M   5210.3;
      =     M    516.1;
      A     L      0.0;
      BLD   102;
      =     M    516.7;
NETWORK
TITLE =

      A     M   1000.0;
      A     I    152.2;
      A     M   5100.2;
      A     M   5110.2;
      A     M   5200.2;
      A     M   5210.2;
      =     M    516.2;
NETWORK
TITLE =

      A     M   1000.6;
      A     M   1500.6;
      A     M   2000.6;
      A     M   5100.1;
      A     M   5110.1;
      A     M   5200.1;
      A     M   5210.1;
      =     M    516.3;
NETWORK
TITLE =

      A     M   1000.2;
      A     M   1500.2;
      A     M   2000.2;
      A     M   5100.0;
      A     M   5110.0;
      A     M   5200.0;
      A     M   5210.0;
      =     M    516.4;
NETWORK
TITLE =

      AN    M   1003.7;
      AN    M   1503.7;
      AN    M   2003.7;
      AN    M   5103.7;
      AN    M   5113.7;
      AN    M   5203.7;
      AN    M   5213.7;
      NOT   ;
      =     M    516.5;
NETWORK
TITLE =

      A     M   1005.0;
      A     M   5016.0;
      A     M   1505.0;
      A     M   2005.0;
      A     M   5105.0;
      A     M   5115.0;
      A     M   5205.0;
      A     M   5215.0;
      =     M    516.6;
NETWORK
TITLE =

      A     M   1009.0;
      A     M   1508.0;
      A     M   2008.0;
      A     M   5104.0;
      A     M   5114.0;
      A     M   5204.0;
      A     M   5214.0;
      =     M    517.0;
NETWORK
TITLE =

      A     M   1009.1;
      A     M   1508.1;
      A     M   2008.1;
      A     M   5104.1;
      A     M   5114.1;
      A     M   5204.1;
      A     M   5214.1;
      =     M    517.1;
NETWORK
TITLE =

      A     M   1009.6;
      A     M   1508.2;
      A     M   2008.2;
      A     M   5104.2;
      A     M   5114.2;
      A     M   5204.2;
      A     M   5214.2;
      =     M    517.2;
NETWORK
TITLE =

      A     M   1009.7;
      A     M   1508.3;
      A     M   2008.3;
      A     M   5104.3;
      A     M   5114.3;
      A     M   5204.3;
      A     M   5214.3;
      =     M    517.3;
NETWORK
TITLE =
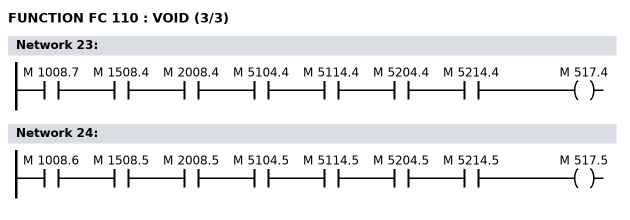

      A     M   1008.7;
      A     M   1508.4;
      A     M   2008.4;
      A     M   5104.4;
      A     M   5114.4;
      A     M   5204.4;
      A     M   5214.4;
      =     M    517.4;
NETWORK
TITLE =

      A     M   1008.6;
      A     M   1508.5;
      A     M   2008.5;
      A     M   5104.5;
      A     M   5114.5;
      A     M   5204.5;
      A     M   5214.5;
      =     M    517.5;
END_FUNCTION

FUNCTION_BLOCK FB 111
TITLE =
VERSION : 0.1

BEGIN
NETWORK
TITLE =
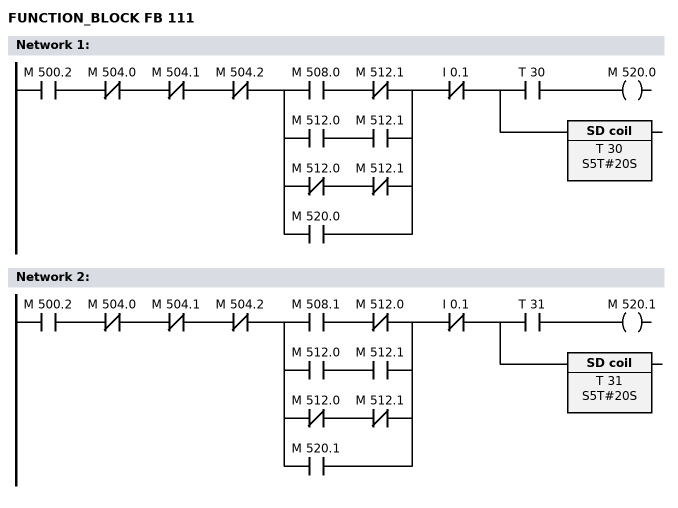

      A     M    500.2;
      AN    M    504.0;
      AN    M    504.1;
      AN    M    504.2;
      A(    ;
      A     M    508.0;
      AN    M    512.1;
      O     ;
      A     M    512.0;
      A     M    512.1;
      O     ;
      AN    M    512.0;
      AN    M    512.1;
      O     M    520.0;
      )     ;
      AN    I      0.1;
      =     L      0.0;
      A     L      0.0;
      A     T     30;
      =     M    520.0;
      A     L      0.0;
      BLD   102;
      L     S5T#20S;
      SD    T     30;
NETWORK
TITLE =

      A     M    500.2;
      AN    M    504.0;
      AN    M    504.1;
      AN    M    504.2;
      A(    ;
      A     M    508.1;
      AN    M    512.0;
      O     ;
      A     M    512.0;
      A     M    512.1;
      O     ;
      AN    M    512.0;
      AN    M    512.1;
      O     M    520.1;
      )     ;
      AN    I      0.1;
      =     L      0.0;
      A     L      0.0;
      A     T     31;
      =     M    520.1;
      A     L      0.0;
      BLD   102;
      L     S5T#20S;
      SD    T     31;
END_FUNCTION_BLOCK

DATA_BLOCK DB 111
TITLE =
VERSION : 0.0

 FB 111
BEGIN
END_DATA_BLOCK

FUNCTION FC 111 : VOID
TITLE =
VERSION : 0.1

BEGIN
NETWORK
TITLE =

      AN    OV;
      =     L      0.0;
      A     L      0.0;
      A     M    508.0;
      A     M    516.6;
      A     M    517.0;
      AN    I     73.1;
      AN    I     73.0;
      S     M    508.6;
      S     M    508.7;
      A     L      0.0;
      A     M    508.1;
      A     M    517.1;
      R     M    508.6;
      A     L      0.0;
      A(    ;
      O     M    512.1;
      O     M    512.0;
      )     ;
      AN    M    517.0;
      R     M    508.7;
END_FUNCTION

FUNCTION_BLOCK FB 112
TITLE =
VERSION : 0.1

BEGIN
NETWORK
TITLE =
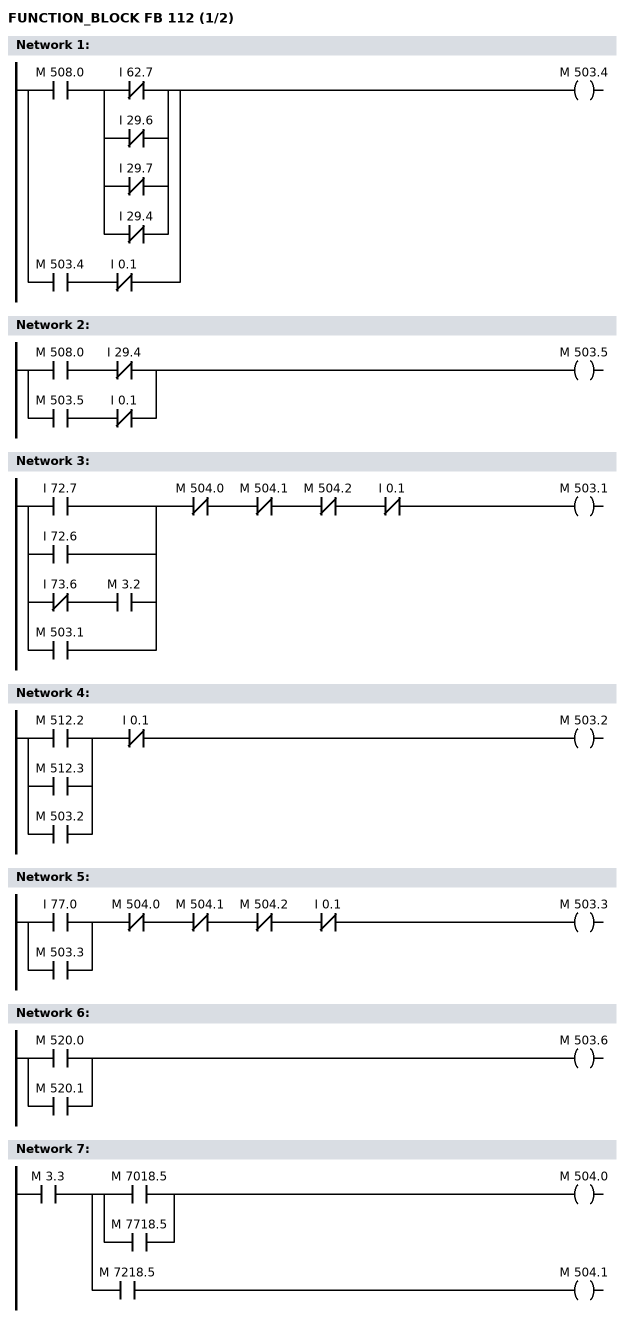

      A     M    508.0;
      A(    ;
      ON    I     62.7;
      ON    I     29.6;
      ON    I     29.7;
      ON    I     29.4;
      )     ;
      O     ;
      A     M    503.4;
      AN    I      0.1;
      =     M    503.4;
NETWORK
TITLE =

      A     M    508.0;
      AN    I     29.4;
      O     ;
      A     M    503.5;
      AN    I      0.1;
      =     M    503.5;
NETWORK
TITLE =

      A(    ;
      O     I     72.7;
      O     I     72.6;
      O     ;
      AN    I     73.6;
      A     M      3.2;
      O     M    503.1;
      )     ;
      AN    M    504.0;
      AN    M    504.1;
      AN    M    504.2;
      AN    I      0.1;
      =     M    503.1;
NETWORK
TITLE =

      A(    ;
      O     M    512.2;
      O     M    512.3;
      O     M    503.2;
      )     ;
      AN    I      0.1;
      =     M    503.2;
NETWORK
TITLE =

      A(    ;
      O     I     77.0;
      O     M    503.3;
      )     ;
      AN    M    504.0;
      AN    M    504.1;
      AN    M    504.2;
      AN    I      0.1;
      =     M    503.3;
NETWORK
TITLE =

      O     M    520.0;
      O     M    520.1;
      =     M    503.6;
NETWORK
TITLE =

      A     M      3.3;
      =     L      0.0;
      A     L      0.0;
      A(    ;
      O     M   7018.5;
      O     M   7718.5;
      )     ;
      =     M    504.0;
      A     L      0.0;
      A     M   7218.5;
      =     M    504.1;
NETWORK
TITLE =
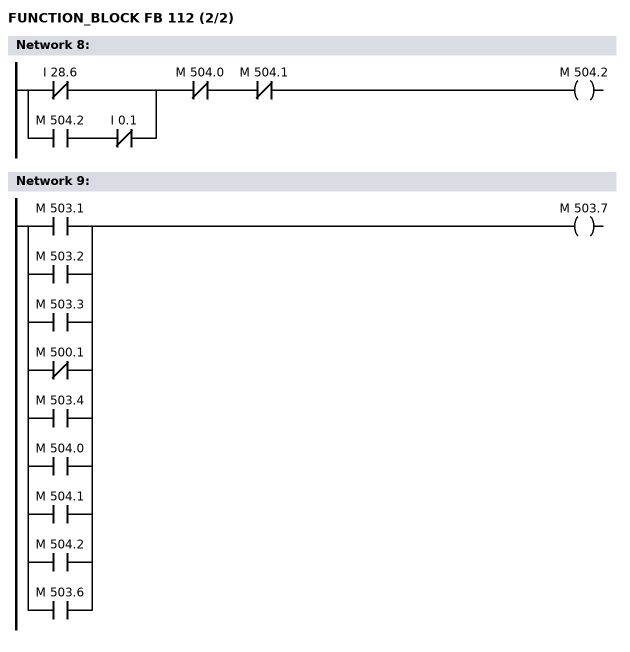

      A(    ;
      ON    I     28.6;
      O     ;
      A     M    504.2;
      AN    I      0.1;
      )     ;
      AN    M    504.0;
      AN    M    504.1;
      =     M    504.2;
NETWORK
TITLE =

      O     M    503.1;
      O     M    503.2;
      O     M    503.3;
      ON    M    500.1;
      O     M    503.4;
      O     M    504.0;
      O     M    504.1;
      O     M    504.2;
      O     M    503.6;
      =     M    503.7;
END_FUNCTION_BLOCK

DATA_BLOCK DB 112
TITLE =
VERSION : 0.0

 FB 112
BEGIN
END_DATA_BLOCK

FUNCTION FC 112 : VOID
TITLE =
VERSION : 0.1

BEGIN
NETWORK
TITLE =
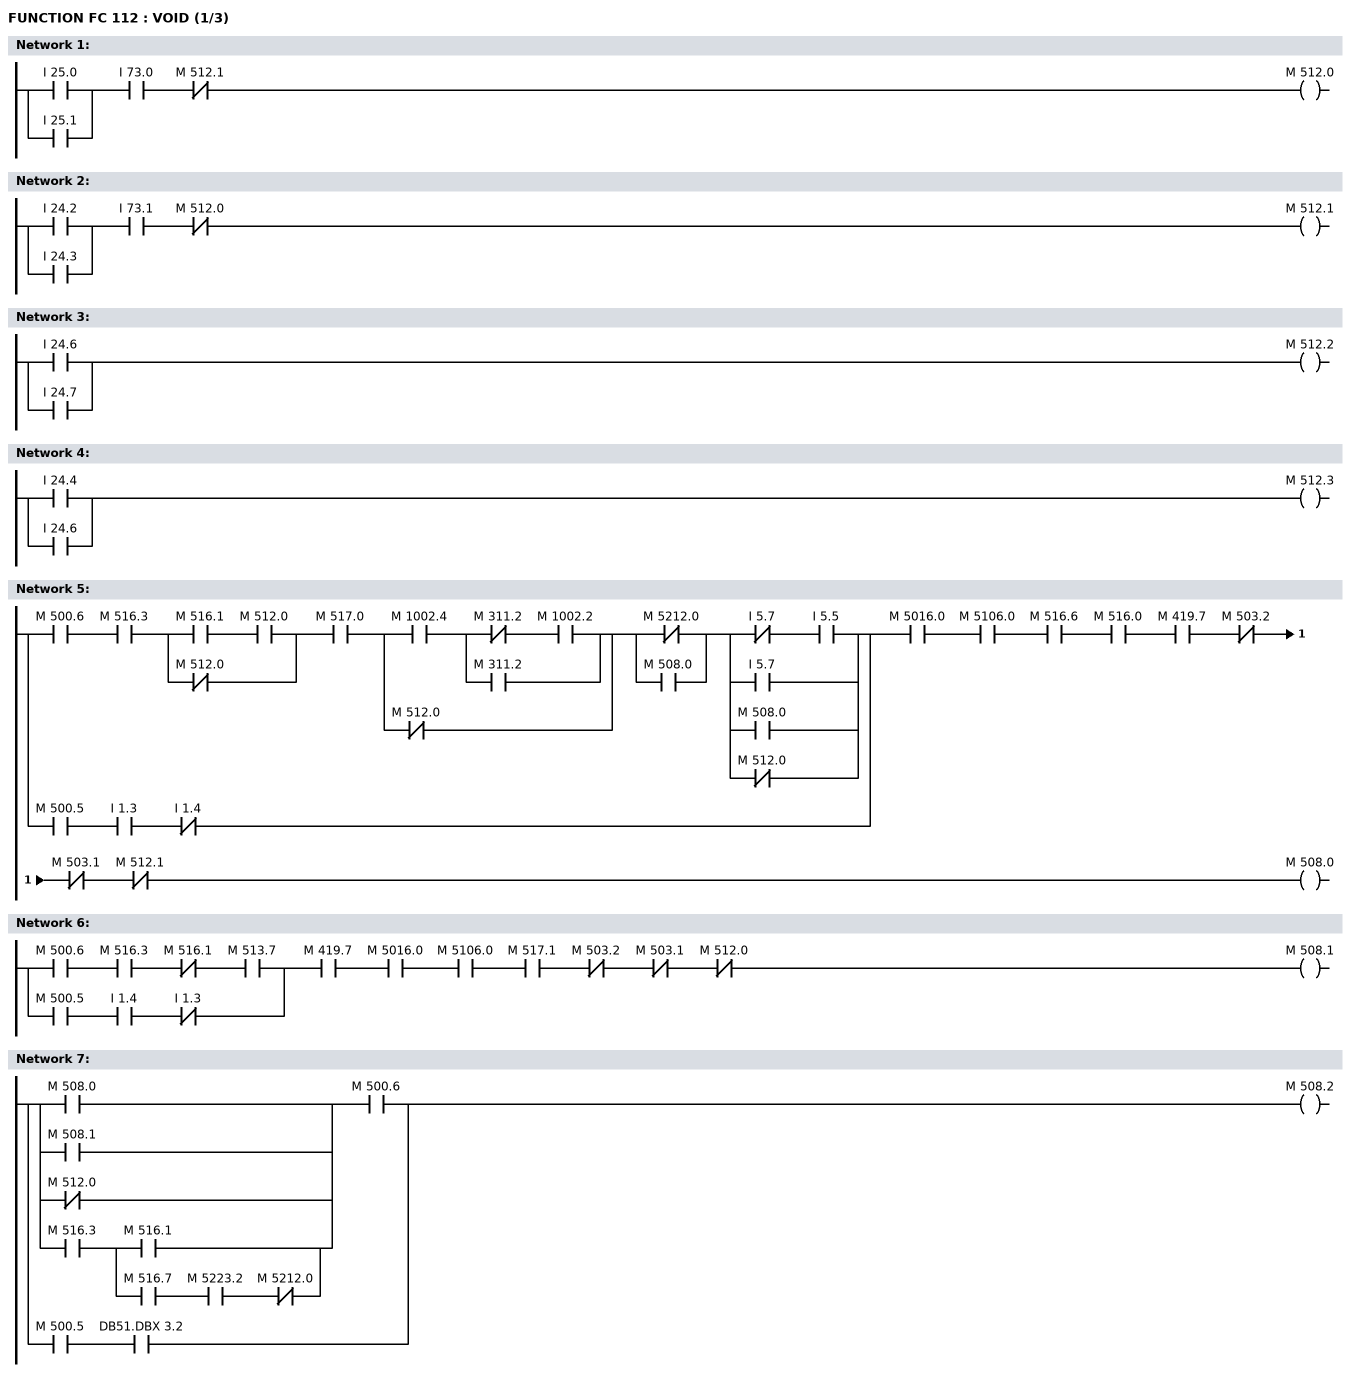

      A(    ;
      O     I     25.0;
      O     I     25.1;
      )     ;
      A     I     73.0;
      AN    M    512.1;
      =     M    512.0;
NETWORK
TITLE =

      A(    ;
      O     I     24.2;
      O     I     24.3;
      )     ;
      A     I     73.1;
      AN    M    512.0;
      =     M    512.1;
NETWORK
TITLE =

      O     I     24.6;
      O     I     24.7;
      =     M    512.2;
NETWORK
TITLE =

      O     I     24.4;
      O     I     24.6;
      =     M    512.3;
NETWORK
TITLE =

      A(    ;
      A     M    500.6;
      A     M    516.3;
      A(    ;
      A     M    516.1;
      A     M    512.0;
      ON    M    512.0;
      )     ;
      A     M    517.0;
      A(    ;
      A     M   1002.4;
      A(    ;
      AN    M    311.2;
      A     M   1002.2;
      O     M    311.2;
      )     ;
      ON    M    512.0;
      )     ;
      A(    ;
      ON    M   5212.0;
      O     M    508.0;
      )     ;
      A(    ;
      AN    I      5.7;
      A     I      5.5;
      O     I      5.7;
      O     M    508.0;
      ON    M    512.0;
      )     ;
      O     ;
      A     M    500.5;
      A     I      1.3;
      AN    I      1.4;
      )     ;
      A     M   5016.0;
      A     M   5106.0;
      A     M    516.6;
      A     M    516.0;
      A     M    419.7;
      AN    M    503.2;
      AN    M    503.1;
      AN    M    512.1;
      =     M    508.0;
NETWORK
TITLE =

      A(    ;
      A     M    500.6;
      A     M    516.3;
      AN    M    516.1;
      A     M    513.7;
      O     ;
      A     M    500.5;
      A     I      1.4;
      AN    I      1.3;
      )     ;
      A     M    419.7;
      A     M   5016.0;
      A     M   5106.0;
      A     M    517.1;
      AN    M    503.2;
      AN    M    503.1;
      AN    M    512.0;
      =     M    508.1;
NETWORK
TITLE =

      A(    ;
      O     M    508.0;
      O     M    508.1;
      ON    M    512.0;
      O     ;
      A     M    516.3;
      A(    ;
      O     M    516.1;
      O     ;
      A     M    516.7;
      A     M   5223.2;
      AN    M   5212.0;
      )     ;
      )     ;
      A     M    500.6;
      O     ;
      A     M    500.5;
      A     DB51.DBX    3.2;
      =     M    508.2;
NETWORK
TITLE =
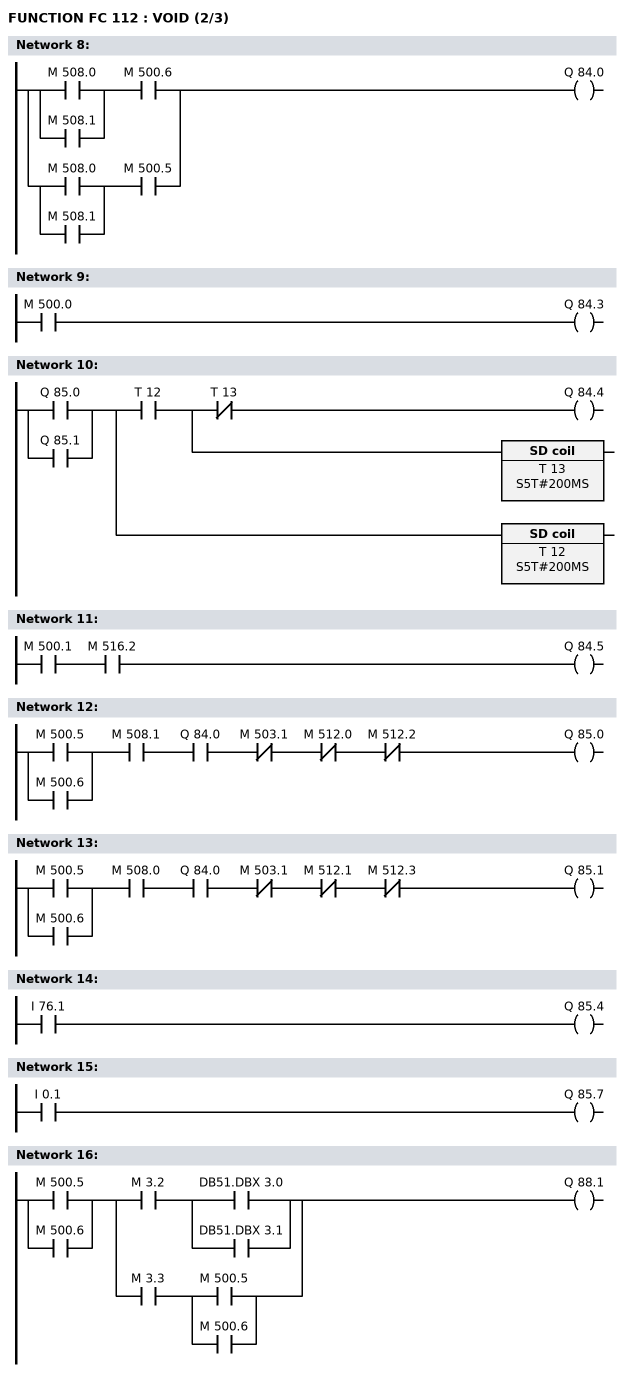

      A(    ;
      O     M    508.0;
      O     M    508.1;
      )     ;
      A     M    500.6;
      O     ;
      A(    ;
      O     M    508.0;
      O     M    508.1;
      )     ;
      A     M    500.5;
      =     Q     84.0;
NETWORK
TITLE =

      A     M    500.0;
      =     Q     84.3;
NETWORK
TITLE =

      O     Q     85.0;
      O     Q     85.1;
      =     L      0.0;
      A     L      0.0;
      A     T     12;
      =     L      0.1;
      A     L      0.1;
      AN    T     13;
      =     Q     84.4;
      A     L      0.1;
      BLD   102;
      L     S5T#200MS;
      SD    T     13;
      A     L      0.0;
      BLD   102;
      L     S5T#200MS;
      SD    T     12;
NETWORK
TITLE =

      A     M    500.1;
      A     M    516.2;
      =     Q     84.5;
NETWORK
TITLE =

      A(    ;
      O     M    500.5;
      O     M    500.6;
      )     ;
      A     M    508.1;
      A     Q     84.0;
      AN    M    503.1;
      AN    M    512.0;
      AN    M    512.2;
      =     Q     85.0;
NETWORK
TITLE =

      A(    ;
      O     M    500.5;
      O     M    500.6;
      )     ;
      A     M    508.0;
      A     Q     84.0;
      AN    M    503.1;
      AN    M    512.1;
      AN    M    512.3;
      =     Q     85.1;
NETWORK
TITLE =

      A     I     76.1;
      =     Q     85.4;
NETWORK
TITLE =

      A     I      0.1;
      =     Q     85.7;
NETWORK
TITLE =

      A(    ;
      O     M    500.5;
      O     M    500.6;
      )     ;
      A(    ;
      A     M      3.2;
      A(    ;
      O     DB51.DBX    3.0;
      O     DB51.DBX    3.1;
      )     ;
      O     ;
      A     M      3.3;
      A(    ;
      O     M    500.5;
      O     M    500.6;
      )     ;
      )     ;
      =     Q     88.1;
NETWORK
TITLE =
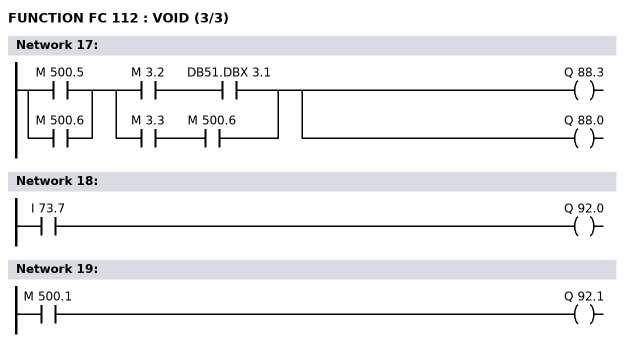

      A(    ;
      O     M    500.5;
      O     M    500.6;
      )     ;
      A(    ;
      A     M      3.2;
      A     DB51.DBX    3.1;
      O     ;
      A     M      3.3;
      A     M    500.6;
      )     ;
      =     Q     88.3;
      =     Q     88.0;
NETWORK
TITLE =

      A     I     73.7;
      =     Q     92.0;
NETWORK
TITLE =

      A     M    500.1;
      =     Q     92.1;
END_FUNCTION

FUNCTION FC 113 : VOID
TITLE =
VERSION : 0.1

BEGIN
NETWORK
TITLE =

      AN    OV;
      =     L      0.0;
      A     L      0.0;
      A(    ;
      O     M   1000.2;
      O     ;
      A     M      0.5;
      AN    M   1000.2;
      )     ;
      =     Q    168.0;
      A     L      0.0;
      A(    ;
      O     M   1000.6;
      O     ;
      A     M      0.5;
      AN    M   1000.6;
      AN    M   1000.5;
      )     ;
      =     Q    168.1;
      A     L      0.0;
      A     M   1001.1;
      =     Q    168.2;
      A     L      0.0;
      A(    ;
      O     M   1001.0;
      O     ;
      A     T     20;
      AN    M   1001.0;
      A     M      0.5;
      )     ;
      =     Q    168.3;
      A     L      0.0;
      A(    ;
      A     M   1003.7;
      A     M      0.5;
      O     M     80.0;
      )     ;
      =     Q    168.4;
      A     L      0.0;
      A(    ;
      ON    M   1000.0;
      ON    I     17.2;
      )     ;
      A     M      0.5;
      =     Q    168.5;
      A(    ;
      A     L      0.0;
      A     OV;
      JNB   _001;
      L     0;
      T     MW    40;
      SET   ;
      SAVE  ;
      CLR   ;
_001: A     BR;
      )     ;
      JNB   _002;
      CALL SFC   21 (
           BVAL                     := MW    40,
           RET_VAL                  := MW   132,
           BLK                      := P#M 3800.0 BYTE 100);
_002: NOP   0;
NETWORK
TITLE =

      AN    OV;
      =     L      0.0;
      A     L      0.0;
      A(    ;
      O     M   1500.2;
      O     ;
      A     M      0.5;
      AN    M   1500.2;
      )     ;
      =     Q    168.6;
      A     L      0.0;
      A(    ;
      O     M   1500.6;
      O     ;
      A     M      0.5;
      AN    M   1500.6;
      AN    M   1500.5;
      )     ;
      =     Q    168.7;
      A     L      0.0;
      A     M   1501.1;
      =     Q    169.0;
      A     L      0.0;
      A(    ;
      O     M   1501.0;
      O     ;
      A     T     20;
      AN    M   1501.0;
      A     M      0.5;
      )     ;
      =     Q    169.1;
      A     L      0.0;
      A     M   1503.7;
      A     M      0.5;
      =     Q    169.2;
      A     L      0.0;
      AN    M   1500.0;
      A     M      0.5;
      =     Q    169.3;
NETWORK
TITLE =

      AN    OV;
      =     L      0.0;
      A     L      0.0;
      A(    ;
      O     M   2000.2;
      O     ;
      A     M      0.5;
      AN    M   2000.2;
      )     ;
      =     Q    169.4;
      A     L      0.0;
      A(    ;
      O     M   2000.6;
      O     ;
      A     M      0.5;
      AN    M   2000.6;
      AN    M   2000.5;
      )     ;
      =     Q    169.5;
      A     L      0.0;
      A     M   2001.1;
      =     Q    169.6;
      A     L      0.0;
      A(    ;
      O     M   2001.0;
      O     ;
      A     T     20;
      AN    M   2001.0;
      A     M      0.5;
      )     ;
      =     Q    169.7;
      A     L      0.0;
      A(    ;
      A     M   2003.7;
      A     M      0.5;
      O     M     81.0;
      )     ;
      =     Q    170.0;
      A     L      0.0;
      AN    M   2000.0;
      A     M      0.5;
      =     Q    170.1;
NETWORK
TITLE =

      AN    OV;
      =     L      0.0;
      A     L      0.0;
      A(    ;
      O     M   5100.0;
      O     ;
      A     M      0.5;
      AN    M   5100.0;
      )     ;
      =     Q    170.2;
      A     L      0.0;
      A(    ;
      O     M   5100.1;
      O     ;
      A     M      0.5;
      AN    M   5100.1;
      AN    M   5100.5;
      )     ;
      =     Q    170.3;
      A     L      0.0;
      A     M   5100.4;
      =     Q    170.4;
      A     L      0.0;
      A(    ;
      O     M   5100.3;
      O     ;
      A     T     20;
      AN    M   5100.3;
      A     M      0.5;
      )     ;
      =     Q    170.5;
      A     L      0.0;
      A(    ;
      A     M   5103.7;
      A     M      0.5;
      O     M   5111.0;
      )     ;
      =     Q    170.6;
      A     L      0.0;
      A(    ;
      ON    M   5100.2;
      ON    M   5102.1;
      )     ;
      A     M      0.5;
      =     Q    170.7;
NETWORK
TITLE =

      AN    OV;
      =     L      0.0;
      A     L      0.0;
      A(    ;
      O     M   5110.0;
      O     ;
      A     M      0.5;
      AN    M   5110.0;
      )     ;
      =     Q    171.0;
      A     L      0.0;
      A(    ;
      O     M   5110.1;
      O     ;
      A     M      0.5;
      AN    M   5110.1;
      AN    M   5110.5;
      )     ;
      =     Q    171.1;
      A     L      0.0;
      A     M   5110.4;
      =     Q    171.2;
      A     L      0.0;
      A(    ;
      O     M   5110.3;
      O     ;
      A     T     20;
      AN    M   5110.3;
      A     M      0.5;
      )     ;
      =     Q    171.3;
      A     L      0.0;
      A(    ;
      A     M   5113.7;
      A     M      0.5;
      O     M   5111.1;
      )     ;
      =     Q    171.4;
      A     L      0.0;
      A(    ;
      ON    M   5110.2;
      ON    M   5102.1;
      )     ;
      A     M      0.5;
      =     Q    171.5;
NETWORK
TITLE =

      AN    OV;
      =     L      0.0;
      A     L      0.0;
      A(    ;
      O     M   5200.0;
      O     ;
      A     M      0.5;
      AN    M   5200.0;
      )     ;
      =     Q    171.6;
      A     L      0.0;
      A(    ;
      O     M   5200.1;
      O     ;
      A     M      0.5;
      AN    M   5200.1;
      AN    M   5200.5;
      )     ;
      =     Q    171.7;
      A     L      0.0;
      A     M   5200.4;
      =     Q    172.0;
      A     L      0.0;
      A(    ;
      O     M   5200.3;
      O     ;
      A     T     20;
      AN    M   5200.3;
      A     M      0.5;
      )     ;
      =     Q    172.1;
      A     L      0.0;
      A(    ;
      A     M   5203.7;
      A     M      0.5;
      O     ;
      A     M   5111.2;
      AN    M   5111.2;
      )     ;
      =     Q    172.2;
      A     L      0.0;
      A(    ;
      ON    M   5200.2;
      O     M   5203.6;
      )     ;
      A     M      0.5;
      =     Q    172.3;
NETWORK
TITLE =

      AN    OV;
      =     L      0.0;
      A     L      0.0;
      A(    ;
      O     M   5210.0;
      O     ;
      A     M      0.5;
      AN    M   5210.0;
      )     ;
      =     Q    172.4;
      A     L      0.0;
      A(    ;
      O     M   5210.1;
      O     ;
      A     M      0.5;
      AN    M   5210.1;
      AN    M   5210.5;
      )     ;
      =     Q    172.5;
      A     L      0.0;
      A(    ;
      A     M   5210.4;
      AN    M   5212.0;
      O     ;
      A     M   5210.4;
      A     M   5212.0;
      A     M      0.5;
      )     ;
      =     Q    172.6;
      A     L      0.0;
      A(    ;
      O     M   5210.3;
      O     ;
      A     T     20;
      AN    M   5210.3;
      A     M      0.5;
      )     ;
      =     Q    172.7;
      A     L      0.0;
      A     M   5213.7;
      A     M      0.5;
      =     Q    173.0;
      A     L      0.0;
      A(    ;
      ON    M   5210.2;
      O     M   5203.6;
      )     ;
      A     M      0.5;
      =     Q    173.1;
NETWORK
TITLE =

      AN    OV;
      =     L      0.0;
      A     L      0.0;
      A(    ;
      O     M    500.2;
      O     ;
      A     M      0.5;
      AN    M    500.2;
      )     ;
      =     Q    173.2;
      A     L      0.0;
      A(    ;
      O     M    500.6;
      O     ;
      A     M      0.5;
      AN    M    500.6;
      AN    M    500.5;
      )     ;
      =     Q    173.3;
      A     L      0.0;
      A     M    517.1;
      =     Q    173.4;
      A     L      0.0;
      A     M    517.0;
      =     Q    173.5;
      A     L      0.0;
      A     M    512.0;
      =     Q    173.6;
      A     L      0.0;
      A     M    512.1;
      =     Q    173.7;
      A     L      0.0;
      A     M    503.7;
      A     M      0.5;
      =     Q    174.0;
      A     L      0.0;
      AN    M    500.1;
      A     M      0.5;
      =     Q    174.1;
NETWORK
TITLE =

      AN    OV;
      =     L      0.0;
      A     L      0.0;
      A     M    516.3;
      =     Q    174.2;
      A     L      0.0;
      A     M    516.5;
      =     Q    174.3;
      A     L      0.0;
      A(    ;
      O     I      2.5;
      O     T     20;
      )     ;
      =     Q    174.4;
NETWORK
TITLE =
